LIN {X 0,Y 368.091,Z 174.068,A -85,B 0,C 180,E1 -12913.968,E2 -12913.968} C_VEL
LIN {X 0,Y 364.016,Z 163.404,A -85,B 0,C 180,E1 -12914.51,E2 -12914.51} C_VEL
LIN {X 0,Y 361.954,Z 153.4,A -85,B 0,C 180,E1 -12917.362,E2 -12917.362} C_VEL
LIN {X 0,Y 361.871,Z 153.409,A -85,B 0,C 180,E1 -12920.973,E2 -12920.973} C_VEL
LIN {X 0,Y 361.871,Z 153.409,A -85,B 0,C 180,E1 -12924.656,E2 -12924.656} C_VEL
LIN {X 0,Y 361.835,Z 153.411,A -85,B 0,C 180,E1 -12928.372,E2 -12928.372} C_VEL
LIN {X 0,Y 361.898,Z 153.403,A -85,B 0,C 180,E1 -12930.956,E2 -12930.956} C_VEL
LIN {X 0,Y 361.953,Z 153.4,A -85,B 0,C 180,E1 -12933.476,E2 -12933.476} C_VEL
LIN {X 0,Y 361.889,Z 153.41,A -85,B 0,C 180,E1 -12937.146,E2 -12937.146} C_VEL
LIN {X 0,Y 361.903,Z 153.406,A -85,B 0,C 180,E1 -12940.724,E2 -12940.724} C_VEL
LIN {X 0,Y 361.943,Z 153.398,A -85,B 0,C 180,E1 -12944.227,E2 -12944.227} C_VEL
LIN {X 0,Y 361.999,Z 153.388,A -85,B 0,C 180,E1 -12946.529,E2 -12946.529} C_VEL
LIN {X 0,Y 362.001,Z 153.389,A -85,B 0,C 180,E1 -12949.938,E2 -12949.938} C_VEL
LIN {X 0,Y 362.136,Z 153.373,A -85,B 0,C 180,E1 -12953.314,E2 -12953.314} C_VEL
LIN {X 0,Y 362.279,Z 153.352,A -85,B 0,C 180,E1 -12957.777,E2 -12957.777} C_VEL
LIN {X 0,Y 362.382,Z 153.337,A -85,B 0,C 180,E1 -12960.001,E2 -12960.001} C_VEL
LIN {X 0,Y 362.267,Z 153.352,A -85,B 0,C 180,E1 -12962.225,E2 -12962.225} C_VEL
LIN {X 0,Y 362.125,Z 153.37,A -85,B 0,C 180,E1 -12966.688,E2 -12966.688} C_VEL
LIN {X 0,Y 362.001,Z 153.384,A -85,B 0,C 180,E1 -12970.064,E2 -12970.064} C_VEL
LIN {X 0,Y 361.984,Z 153.397,A -85,B 0,C 180,E1 -12973.889,E2 -12973.889} C_VEL
LIN {X 0,Y 361.909,Z 153.405,A -85,B 0,C 180,E1 -12978.103,E2 -12978.103} C_VEL
LIN {X 0,Y 361.855,Z 153.403,A -85,B 0,C 180,E1 -12981.656,E2 -12981.656} C_VEL
LIN {X 0,Y 361.862,Z 153.407,A -85,B 0,C 180,E1 -12985.296,E2 -12985.296} C_VEL
LIN {X 0,Y 361.858,Z 153.411,A -85,B 0,C 180,E1 -12989.074,E2 -12989.074} C_VEL
LIN {X 0,Y 361.849,Z 153.412,A -85,B 0,C 180,E1 -12992.946,E2 -12992.946} C_VEL
LIN {X 0,Y 361.865,Z 153.41,A -85,B 0,C 180,E1 -12995.638,E2 -12995.638} C_VEL
LIN {X 0,Y 361.826,Z 153.414,A -85,B 0,C 180,E1 -12999.018,E2 -12999.018} C_VEL
LIN {X 0,Y 361.831,Z 153.419,A -85,B 0,C 180,E1 -13002.831,E2 -13002.831} C_VEL
LIN {X 0,Y 361.816,Z 153.419,A -85,B 0,C 180,E1 -13005.948,E2 -13005.948} C_VEL
LIN {X 0,Y 361.813,Z 153.419,A -85,B 0,C 180,E1 -13009.25,E2 -13009.25} C_VEL
LIN {X 0,Y 361.866,Z 153.403,A -85,B 0,C 180,E1 -13012.982,E2 -13012.982} C_VEL
LIN {X 0,Y 361.861,Z 153.408,A -85,B 0,C 180,E1 -13016.631,E2 -13016.631} C_VEL
LIN {X 0,Y 361.91,Z 153.464,A -85,B 0,C 180,E1 -13019.485,E2 -13019.485} C_VEL
LIN {X 0,Y 364.43,Z 165.067,A -85,B 0,C 180,E1 -13022.513,E2 -13022.513} C_VEL
LIN {X 0,Y 365.971,Z 173.011,A -85,B 0,C 180,E1 -13024.5,E2 -13024.5} C_VEL
LIN {X 0,Y 365.06,Z 184.322,A -85,B 0,C 180,E1 -13027.055,E2 -13027.055} C_VEL
LIN {X 0,Y 364.787,Z 186.723,A -85,B 0,C 180,E1 -13027.588,E2 -13027.588} C_VEL
LIN {X 0,Y 368.969,Z 210.144,A -85,B 0,C 180,E1 -13028.388,E2 -13028.388} C_VEL
LIN {X 0,Y 370.637,Z 222.589,A -85,B 0,C 180,E1 -13028.758,E2 -13028.758} C_VEL
LIN {X 0,Y 369.343,Z 296.316,A -85,B 0,C 180,E1 -13030.26,E2 -13030.26} C_VEL
LIN {X 0,Y 368.516,Z 309.974,A -85,B 0,C 180,E1 -13030.757,E2 -13030.757} C_VEL
LIN {X 0,Y 367.539,Z 322.813,A -85,B 0,C 180,E1 -13031.464,E2 -13031.464} C_VEL
LIN {X 0,Y 366.451,Z 335.344,A -85,B 0,C 180,E1 -13032.419,E2 -13032.419} C_VEL
LIN {X 0,Y 365.246,Z 346.544,A -85,B 0,C 180,E1 -13033.512,E2 -13033.512} C_VEL
LIN {X 0,Y 364.166,Z 356.855,A -85,B 0,C 180,E1 -13034.786,E2 -13034.786} C_VEL
LIN {X 0,Y 363.107,Z 366.602,A -85,B 0,C 180,E1 -13036.285,E2 -13036.285} C_VEL
LIN {X 0,Y 362.031,Z 375.393,A -85,B 0,C 180,E1 -13037.955,E2 -13037.955} C_VEL
LIN {X 0,Y 361.31,Z 382.419,A -85,B 0,C 180,E1 -13039.635,E2 -13039.635} C_VEL
LIN {X 0,Y 360.762,Z 388.878,A -85,B 0,C 180,E1 -13041.599,E2 -13041.599} C_VEL
LIN {X 0,Y 360.488,Z 393.134,A -85,B 0,C 180,E1 -13043.283,E2 -13043.283} C_VEL
LIN {X 0,Y 360.348,Z 395.396,A -85,B 0,C 180,E1 -13044.404,E2 -13044.404} C_VEL
LIN {X 0,Y 360.36,Z 397.178,A -85,B 0,C 180,E1 -13045.526,E2 -13045.526} C_VEL
LIN {X 0,Y 360.299,Z 399.5,A -85,B 0,C 180,E1 -13047.764,E2 -13047.764} C_VEL
LIN {X 0,Y 360.371,Z 400.07,A -85,B 0,C 180,E1 -13048.883,E2 -13048.883} C_VEL
LIN {X 0,Y 360.428,Z 400.201,A -85,B 0,C 180,E1 -13050,E2 -13050} C_VEL
LIN {X 0,Y 360.387,Z 399.931,A -85,B 0,C 180,E1 -13051.118,E2 -13051.118} C_VEL
LIN {X 0,Y 360.304,Z 398.214,A -85,B 0,C 180,E1 -13053.355,E2 -13053.355} C_VEL
LIN {X 0,Y 360.36,Z 396.702,A -85,B 0,C 180,E1 -13054.474,E2 -13054.474} C_VEL
LIN {X 0,Y 360.38,Z 394.055,A -85,B 0,C 180,E1 -13055.961,E2 -13055.961} C_VEL
LIN {X 0,Y 360.647,Z 389.498,A -85,B 0,C 180,E1 -13057.84,E2 -13057.84} C_VEL
LIN {X 0,Y 361.077,Z 383.159,A -85,B 0,C 180,E1 -13059.806,E2 -13059.806} C_VEL
LIN {X 0,Y 361.657,Z 376.253,A -85,B 0,C 180,E1 -13061.49,E2 -13061.49} C_VEL
LIN {X 0,Y 362.63,Z 367.626,A -85,B 0,C 180,E1 -13063.163,E2 -13063.163} C_VEL
LIN {X 0,Y 363.61,Z 357.664,A -85,B 0,C 180,E1 -13064.712,E2 -13064.712} C_VEL
LIN {X 0,Y 364.497,Z 347.838,A -85,B 0,C 180,E1 -13065.948,E2 -13065.948} C_VEL
LIN {X 0,Y 365.582,Z 336.839,A -85,B 0,C 180,E1 -13067.048,E2 -13067.048} C_VEL
LIN {X 0,Y 366.652,Z 324.514,A -85,B 0,C 180,E1 -13068.004,E2 -13068.004} C_VEL
LIN {X 0,Y 367.503,Z 312.873,A -85,B 0,C 180,E1 -13068.683,E2 -13068.683} C_VEL
LIN {X 0,Y 368.158,Z 300.549,A -85,B 0,C 180,E1 -13069.19,E2 -13069.19} C_VEL
LIN {X 0,Y 368.573,Z 285.008,A -85,B 0,C 180,E1 -13069.566,E2 -13069.566} C_VEL
LIN {X 0,Y 369.542,Z 221.072,A -85,B 0,C 180,E1 -13070.833,E2 -13070.833} C_VEL
LIN {X 0,Y 364.298,Z 187.546,A -85,B 0,C 180,E1 -13071.838,E2 -13071.838} C_VEL
LIN {X 0,Y 365.573,Z 174.668,A -85,B 0,C 180,E1 -13074.717,E2 -13074.717} C_VEL
LIN {X 0,Y 365.598,Z 171.805,A -85,B 0,C 180,E1 -13075.377,E2 -13075.377} C_VEL
LIN {X 0,Y 363.305,Z 160.054,A -85,B 0,C 180,E1 -13078.291,E2 -13078.291} C_VEL
LIN {X 0,Y 361.879,Z 153.41,A -85,B 0,C 180,E1 -13080.025,E2 -13080.025} C_VEL
LIN {X 0,Y 361.863,Z 153.41,A -85,B 0,C 180,E1 -13083.369,E2 -13083.369} C_VEL
LIN {X 0,Y 361.869,Z 153.407,A -85,B 0,C 180,E1 -13087.018,E2 -13087.018} C_VEL
LIN {X 0,Y 361.816,Z 153.413,A -85,B 0,C 180,E1 -13090.751,E2 -13090.751} C_VEL
LIN {X 0,Y 361.816,Z 153.412,A -85,B 0,C 180,E1 -13094.369,E2 -13094.369} C_VEL
LIN {X 0,Y 361.834,Z 153.413,A -85,B 0,C 180,E1 -13097.569,E2 -13097.569} C_VEL
LIN {X 0,Y 361.849,Z 153.41,A -85,B 0,C 180,E1 -13101.572,E2 -13101.572} C_VEL
LIN {X 0,Y 361.875,Z 153.407,A -85,B 0,C 180,E1 -13104.656,E2 -13104.656} C_VEL
LIN {X 0,Y 361.842,Z 153.41,A -85,B 0,C 180,E1 -13108.37,E2 -13108.37} C_VEL
LIN {X 0,Y 361.871,Z 153.411,A -85,B 0,C 180,E1 -13110.952,E2 -13110.952} C_VEL
LIN {X 0,Y 361.886,Z 153.408,A -85,B 0,C 180,E1 -13114.706,E2 -13114.706} C_VEL
LIN {X 0,Y 361.859,Z 153.409,A -85,B 0,C 180,E1 -13118.344,E2 -13118.344} C_VEL
LIN {X 0,Y 361.909,Z 153.402,A -85,B 0,C 180,E1 -13122.092,E2 -13122.092} C_VEL
LIN {X 0,Y 361.985,Z 153.393,A -85,B 0,C 180,E1 -13126.112,E2 -13126.112} C_VEL
LIN {X 0,Y 362.003,Z 153.39,A -85,B 0,C 180,E1 -13129.936,E2 -13129.936} C_VEL
LIN {X 0,Y 362.126,Z 153.374,A -85,B 0,C 180,E1 -13133.312,E2 -13133.312} C_VEL
LIN {X 0,Y 362.268,Z 153.357,A -85,B 0,C 180,E1 -13137.775,E2 -13137.775} C_VEL
LIN {X 0,Y 362.179,Z 153.367,A -85,B 0,C 180,E1 -13141.111,E2 -13141.111} C_VEL
LIN {X 0,Y 362.267,Z 153.362,A -85,B 0,C 180,E1 -13142.223,E2 -13142.223} C_VEL
LIN {X 0,Y 362.122,Z 153.375,A -85,B 0,C 180,E1 -13146.686,E2 -13146.686} C_VEL
LIN {X 0,Y 361.997,Z 153.395,A -85,B 0,C 180,E1 -13150.062,E2 -13150.062} C_VEL
LIN {X 0,Y 361.982,Z 153.398,A -85,B 0,C 180,E1 -13153.886,E2 -13153.886} C_VEL
LIN {X 0,Y 361.885,Z 153.407,A -85,B 0,C 180,E1 -13158.102,E2 -13158.102} C_VEL
LIN {X 0,Y 361.853,Z 153.413,A -85,B 0,C 180,E1 -13161.654,E2 -13161.654} C_VEL
LIN {X 0,Y 361.852,Z 153.411,A -85,B 0,C 180,E1 -13165.295,E2 -13165.295} C_VEL
LIN {X 0,Y 361.855,Z 153.409,A -85,B 0,C 180,E1 -13169.072,E2 -13169.072} C_VEL
LIN {X 0,Y 361.846,Z 153.41,A -85,B 0,C 180,E1 -13172.944,E2 -13172.944} C_VEL
LIN {X 0,Y 361.865,Z 153.41,A -85,B 0,C 180,E1 -13175.636,E2 -13175.636} C_VEL
LIN {X 0,Y 361.823,Z 153.415,A -85,B 0,C 180,E1 -13179.017,E2 -13179.017} C_VEL
LIN {X 0,Y 361.827,Z 153.413,A -85,B 0,C 180,E1 -13182.829,E2 -13182.829} C_VEL
LIN {X 0,Y 361.809,Z 153.413,A -85,B 0,C 180,E1 -13185.946,E2 -13185.946} C_VEL
LIN {X 0,Y 361.808,Z 153.417,A -85,B 0,C 180,E1 -13189.248,E2 -13189.248} C_VEL
LIN {X 0,Y 361.858,Z 153.413,A -85,B 0,C 180,E1 -13192.98,E2 -13192.98} C_VEL
LIN {X 0,Y 361.852,Z 153.411,A -85,B 0,C 180,E1 -13196.63,E2 -13196.63} C_VEL
LIN {X 0,Y 361.85,Z 153.408,A -85,B 0,C 180,E1 -13199.669,E2 -13199.669} C_VEL
LIN {X 0,Y 361.849,Z 153.408,A -85,B 0,C 180,E1 -13203.466,E2 -13203.466} C_VEL
LIN {X 0,Y 361.855,Z 153.409,A -85,B 0,C 180,E1 -13207.142,E2 -13207.142} C_VEL
LIN {X 0,Y 361.847,Z 153.413,A -85,B 0,C 180,E1 -13210.72,E2 -13210.72} C_VEL
LIN {X 0,Y 361.888,Z 153.407,A -85,B 0,C 180,E1 -13214.223,E2 -13214.223} C_VEL
LIN {X 0,Y 361.992,Z 153.395,A -85,B 0,C 180,E1 -13216.527,E2 -13216.527} C_VEL
LIN {X 0,Y 361.987,Z 153.393,A -85,B 0,C 180,E1 -13219.936,E2 -13219.936} C_VEL
LIN {X 0,Y 362.114,Z 153.375,A -85,B 0,C 180,E1 -13223.312,E2 -13223.312} C_VEL
LIN {X 0,Y 362.189,Z 153.39,A -85,B 0,C 180,E1 -13227.567,E2 -13227.567} C_VEL
LIN {X 0,Y 363.918,Z 163.048,A -85,B 0,C 180,E1 -13230.214,E2 -13230.214} C_VEL
LIN {X 0,Y 366.792,Z 172.146,A -85,B 0,C 180,E1 -13230.576,E2 -13230.576} C_VEL
LIN {X 0,Y 370.036,Z 187.803,A -85,B 0,C 180,E1 -13231.088,E2 -13231.088} C_VEL
LIN {X 0,Y 368.599,Z 270.026,A -85,B 0,C 180,E1 -13232.732,E2 -13232.732} C_VEL
LIN {X 0,Y 368.077,Z 282.649,A -85,B 0,C 180,E1 -13233.181,E2 -13233.181} C_VEL
LIN {X 0,Y 367.405,Z 296.158,A -85,B 0,C 180,E1 -13233.907,E2 -13233.907} C_VEL
LIN {X 0,Y 366.547,Z 308.584,A -85,B 0,C 180,E1 -13234.834,E2 -13234.834} C_VEL
LIN {X 0,Y 365.609,Z 319.937,A -85,B 0,C 180,E1 -13235.93,E2 -13235.93} C_VEL
LIN {X 0,Y 364.589,Z 330.413,A -85,B 0,C 180,E1 -13237.198,E2 -13237.198} C_VEL
LIN {X 0,Y 363.606,Z 339.787,A -85,B 0,C 180,E1 -13238.615,E2 -13238.615} C_VEL
LIN {X 0,Y 362.596,Z 348.911,A -85,B 0,C 180,E1 -13240.328,E2 -13240.328} C_VEL
LIN {X 0,Y 361.859,Z 356.191,A -85,B 0,C 180,E1 -13242.051,E2 -13242.051} C_VEL
LIN {X 0,Y 361.331,Z 361.133,A -85,B 0,C 180,E1 -13243.497,E2 -13243.497} C_VEL
LIN {X 0,Y 360.906,Z 365.868,A -85,B 0,C 180,E1 -13245.241,E2 -13245.241} C_VEL
LIN {X 0,Y 360.511,Z 369.794,A -85,B 0,C 180,E1 -13247.213,E2 -13247.213} C_VEL
LIN {X 0,Y 360.275,Z 372.567,A -85,B 0,C 180,E1 -13249.367,E2 -13249.367} C_VEL
LIN {X 0,Y 360.162,Z 373.608,A -85,B 0,C 180,E1 -13251.025,E2 -13251.025} C_VEL
LIN {X 0,Y 360.2,Z 373.839,A -85,B 0,C 180,E1 -13252.969,E2 -13252.969} C_VEL
LIN {X 0,Y 360.25,Z 373.344,A -85,B 0,C 180,E1 -13254.185,E2 -13254.185} C_VEL
LIN {X 0,Y 360.427,Z 371.817,A -85,B 0,C 180,E1 -13255.879,E2 -13255.879} C_VEL
LIN {X 0,Y 359.904,Z 370.713,A -85,B 0,C 180,E1 -13256.798,E2 -13256.798} C_VEL
LIN {X 0,Y 357.295,Z 368.435,A -85,B 0,C 180,E1 -13258.286,E2 -13258.286} C_VEL
LIN {X 0,Y 355.141,Z 366.13,A -85,B 0,C 180,E1 -13259.465,E2 -13259.465} C_VEL
LIN {X 0,Y 354.359,Z 364.018,A -85,B 0,C 180,E1 -13260.351,E2 -13260.351} C_VEL
LIN {X 0,Y 354.374,Z 363.21,A -85,B 0,C 180,E1 -13260.644,E2 -13260.644} C_VEL
LIN {X 0,Y 355.171,Z 356.911,A -85,B 0,C 180,E1 -13262.63,E2 -13262.63} C_VEL
LIN {X 0,Y 356.081,Z 349.885,A -85,B 0,C 180,E1 -13264.36,E2 -13264.36} C_VEL
LIN {X 0,Y 357.002,Z 342.397,A -85,B 0,C 180,E1 -13265.85,E2 -13265.85} C_VEL
LIN {X 0,Y 358.233,Z 332.376,A -85,B 0,C 180,E1 -13267.458,E2 -13267.458} C_VEL
LIN {X 0,Y 359.421,Z 322.449,A -85,B 0,C 180,E1 -13268.735,E2 -13268.735} C_VEL
LIN {X 0,Y 360.491,Z 311.509,A -85,B 0,C 180,E1 -13269.86,E2 -13269.86} C_VEL
LIN {X 0,Y 361.527,Z 299.931,A -85,B 0,C 180,E1 -13270.789,E2 -13270.789} C_VEL
LIN {X 0,Y 362.271,Z 287.523,A -85,B 0,C 180,E1 -13271.547,E2 -13271.547} C_VEL
LIN {X 0,Y 362.862,Z 274.421,A -85,B 0,C 180,E1 -13272.092,E2 -13272.092} C_VEL
LIN {X 0,Y 363.358,Z 256.473,A -85,B 0,C 180,E1 -13272.513,E2 -13272.513} C_VEL
LIN {X 0,Y 364.736,Z 190.027,A -85,B 0,C 180,E1 -13273.854,E2 -13273.854} C_VEL
LIN {X 0,Y 361.911,Z 176.606,A -85,B 0,C 180,E1 -13274.345,E2 -13274.345} C_VEL
LIN {X 0,Y 356.896,Z 163.731,A -85,B 0,C 180,E1 -13275.013,E2 -13275.013} C_VEL
LIN {X 0,Y 354.874,Z 154.284,A -85,B 0,C 180,E1 -13277.754,E2 -13277.754} C_VEL
LIN {X 0,Y 354.833,Z 154.286,A -85,B 0,C 180,E1 -13280.67,E2 -13280.67} C_VEL
LIN {X 0,Y 354.819,Z 154.289,A -85,B 0,C 180,E1 -13284.302,E2 -13284.302} C_VEL
LIN {X 0,Y 354.784,Z 154.292,A -85,B 0,C 180,E1 -13287.668,E2 -13287.668} C_VEL
LIN {X 0,Y 354.866,Z 154.277,A -85,B 0,C 180,E1 -13290.622,E2 -13290.622} C_VEL
LIN {X 0,Y 354.898,Z 154.279,A -85,B 0,C 180,E1 -13294.174,E2 -13294.174} C_VEL
LIN {X 0,Y 354.834,Z 154.286,A -85,B 0,C 180,E1 -13297.895,E2 -13297.895} C_VEL
LIN {X 0,Y 354.889,Z 154.275,A -85,B 0,C 180,E1 -13301.909,E2 -13301.909} C_VEL
LIN {X 0,Y 354.943,Z 154.267,A -85,B 0,C 180,E1 -13305.982,E2 -13305.982} C_VEL
LIN {X 0,Y 354.957,Z 154.267,A -85,B 0,C 180,E1 -13309.736,E2 -13309.736} C_VEL
LIN {X 0,Y 355.1,Z 154.25,A -85,B 0,C 180,E1 -13313.181,E2 -13313.181} C_VEL
LIN {X 0,Y 355.242,Z 154.229,A -85,B 0,C 180,E1 -13317.733,E2 -13317.733} C_VEL
LIN {X 0,Y 355.333,Z 154.215,A -85,B 0,C 180,E1 -13320.001,E2 -13320.001} C_VEL
LIN {X 0,Y 355.229,Z 154.229,A -85,B 0,C 180,E1 -13322.269,E2 -13322.269} C_VEL
LIN {X 0,Y 355.091,Z 154.247,A -85,B 0,C 180,E1 -13326.821,E2 -13326.821} C_VEL
LIN {X 0,Y 354.957,Z 154.259,A -85,B 0,C 180,E1 -13330.266,E2 -13330.266} C_VEL
LIN {X 0,Y 354.929,Z 154.275,A -85,B 0,C 180,E1 -13334.009,E2 -13334.009} C_VEL
LIN {X 0,Y 354.865,Z 154.282,A -85,B 0,C 180,E1 -13338.079,E2 -13338.079} C_VEL
LIN {X 0,Y 354.808,Z 154.283,A -85,B 0,C 180,E1 -13342.109,E2 -13342.109} C_VEL
LIN {X 0,Y 354.801,Z 154.281,A -85,B 0,C 180,E1 -13345.836,E2 -13345.836} C_VEL
LIN {X 0,Y 354.795,Z 154.285,A -85,B 0,C 180,E1 -13349.685,E2 -13349.685} C_VEL
LIN {X 0,Y 354.788,Z 154.29,A -85,B 0,C 180,E1 -13352.334,E2 -13352.334} C_VEL
LIN {X 0,Y 354.82,Z 154.288,A -85,B 0,C 180,E1 -13355.699,E2 -13355.699} C_VEL
LIN {X 0,Y 354.771,Z 154.297,A -85,B 0,C 180,E1 -13359.413,E2 -13359.413} C_VEL
LIN {X 0,Y 354.783,Z 154.298,A -85,B 0,C 180,E1 -13362.866,E2 -13362.866} C_VEL
LIN {X 0,Y 354.765,Z 154.298,A -85,B 0,C 180,E1 -13366.103,E2 -13366.103} C_VEL
LIN {X 0,Y 354.765,Z 154.297,A -85,B 0,C 180,E1 -13369.176,E2 -13369.176} C_VEL
LIN {X 0,Y 354.803,Z 154.288,A -85,B 0,C 180,E1 -13372.405,E2 -13372.405} C_VEL
LIN {X 0,Y 354.814,Z 154.289,A -85,B 0,C 180,E1 -13374.941,E2 -13374.941} C_VEL
LIN {X 0,Y 354.793,Z 154.288,A -85,B 0,C 180,E1 -13378.407,E2 -13378.407} C_VEL
LIN {X 0,Y 354.842,Z 154.331,A -85,B 0,C 180,E1 -13379.051,E2 -13379.051} C_VEL
LIN {X 0,Y 357.162,Z 164.602,A -85,B 0,C 180,E1 -13381.819,E2 -13381.819} C_VEL
LIN {X 0,Y 359.121,Z 175.083,A -85,B 0,C 180,E1 -13384.498,E2 -13384.498} C_VEL
LIN {X 0,Y 358.055,Z 186.716,A -85,B 0,C 180,E1 -13387.128,E2 -13387.128} C_VEL
LIN {X 0,Y 362.525,Z 211.613,A -85,B 0,C 180,E1 -13387.991,E2 -13387.991} C_VEL
LIN {X 0,Y 364.09,Z 223.708,A -85,B 0,C 180,E1 -13388.357,E2 -13388.357} C_VEL
LIN {X 0,Y 362.74,Z 295.788,A -85,B 0,C 180,E1 -13389.848,E2 -13389.848} C_VEL
LIN {X 0,Y 361.925,Z 309.526,A -85,B 0,C 180,E1 -13390.356,E2 -13390.356} C_VEL
LIN {X 0,Y 360.916,Z 321.914,A -85,B 0,C 180,E1 -13391.038,E2 -13391.038} C_VEL
LIN {X 0,Y 359.832,Z 333.796,A -85,B 0,C 180,E1 -13391.937,E2 -13391.937} C_VEL
LIN {X 0,Y 358.558,Z 345.229,A -85,B 0,C 180,E1 -13393.049,E2 -13393.049} C_VEL
LIN {X 0,Y 357.418,Z 355.6,A -85,B 0,C 180,E1 -13394.319,E2 -13394.319} C_VEL
LIN {X 0,Y 356.353,Z 364.852,A -85,B 0,C 180,E1 -13395.728,E2 -13395.728} C_VEL
LIN {X 0,Y 355.259,Z 373.891,A -85,B 0,C 180,E1 -13397.431,E2 -13397.431} C_VEL
LIN {X 0,Y 354.388,Z 381.186,A -85,B 0,C 180,E1 -13399.141,E2 -13399.141} C_VEL
LIN {X 0,Y 353.855,Z 387.036,A -85,B 0,C 180,E1 -13400.858,E2 -13400.858} C_VEL
LIN {X 0,Y 353.466,Z 391.652,A -85,B 0,C 180,E1 -13402.575,E2 -13402.575} C_VEL
LIN {X 0,Y 353.284,Z 395.175,A -85,B 0,C 180,E1 -13404.292,E2 -13404.292} C_VEL
LIN {X 0,Y 353.27,Z 396.946,A -85,B 0,C 180,E1 -13405.436,E2 -13405.436} C_VEL
LIN {X 0,Y 353.224,Z 398.299,A -85,B 0,C 180,E1 -13406.578,E2 -13406.578} C_VEL
LIN {X 0,Y 353.271,Z 399.816,A -85,B 0,C 180,E1 -13408.86,E2 -13408.86} C_VEL
LIN {X 0,Y 353.332,Z 399.938,A -85,B 0,C 180,E1 -13410,E2 -13410} C_VEL
LIN {X 0,Y 353.287,Z 399.661,A -85,B 0,C 180,E1 -13411.14,E2 -13411.14} C_VEL
LIN {X 0,Y 353.225,Z 397.929,A -85,B 0,C 180,E1 -13413.422,E2 -13413.422} C_VEL
LIN {X 0,Y 353.27,Z 396.405,A -85,B 0,C 180,E1 -13414.564,E2 -13414.564} C_VEL
LIN {X 0,Y 353.335,Z 393.322,A -85,B 0,C 180,E1 -13416.28,E2 -13416.28} C_VEL
LIN {X 0,Y 353.573,Z 389.168,A -85,B 0,C 180,E1 -13417.998,E2 -13417.998} C_VEL
LIN {X 0,Y 354.055,Z 382.812,A -85,B 0,C 180,E1 -13420.003,E2 -13420.003} C_VEL
LIN {X 0,Y 354.663,Z 375.885,A -85,B 0,C 180,E1 -13421.719,E2 -13421.719} C_VEL
LIN {X 0,Y 355.656,Z 367.22,A -85,B 0,C 180,E1 -13423.426,E2 -13423.426} C_VEL
LIN {X 0,Y 356.605,Z 358.323,A -85,B 0,C 180,E1 -13424.845,E2 -13424.845} C_VEL
LIN {X 0,Y 357.509,Z 348.548,A -85,B 0,C 180,E1 -13426.122,E2 -13426.122} C_VEL
LIN {X 0,Y 358.628,Z 337.858,A -85,B 0,C 180,E1 -13427.242,E2 -13427.242} C_VEL
LIN {X 0,Y 359.718,Z 325.882,A -85,B 0,C 180,E1 -13428.216,E2 -13428.216} C_VEL
LIN {X 0,Y 360.691,Z 313.433,A -85,B 0,C 180,E1 -13428.975,E2 -13428.975} C_VEL
LIN {X 0,Y 361.397,Z 300.561,A -85,B 0,C 180,E1 -13429.527,E2 -13429.527} C_VEL
LIN {X 0,Y 361.836,Z 286.962,A -85,B 0,C 180,E1 -13429.871,E2 -13429.871} C_VEL
LIN {X 0,Y 362.851,Z 222.052,A -85,B 0,C 180,E1 -13431.181,E2 -13431.181} C_VEL
LIN {X 0,Y 357.747,Z 189.335,A -85,B 0,C 180,E1 -13432.175,E2 -13432.175} C_VEL
LIN {X 0,Y 357.447,Z 187.262,A -85,B 0,C 180,E1 -13432.255,E2 -13432.255} C_VEL
LIN {X 0,Y 358.643,Z 175.582,A -85,B 0,C 180,E1 -13434.918,E2 -13434.918} C_VEL
LIN {X 0,Y 358.38,Z 171.625,A -85,B 0,C 180,E1 -13435.87,E2 -13435.87} C_VEL
LIN {X 0,Y 356.008,Z 159.615,A -85,B 0,C 180,E1 -13438.925,E2 -13438.925} C_VEL
LIN {X 0,Y 354.843,Z 154.288,A -85,B 0,C 180,E1 -13440.335,E2 -13440.335} C_VEL
LIN {X 0,Y 354.811,Z 154.29,A -85,B 0,C 180,E1 -13443.702,E2 -13443.702} C_VEL
LIN {X 0,Y 354.8,Z 154.286,A -85,B 0,C 180,E1 -13446.46,E2 -13446.46} C_VEL
LIN {X 0,Y 354.773,Z 154.296,A -85,B 0,C 180,E1 -13449.412,E2 -13449.412} C_VEL
LIN {X 0,Y 354.787,Z 154.289,A -85,B 0,C 180,E1 -13452.866,E2 -13452.866} C_VEL
LIN {X 0,Y 354.767,Z 154.29,A -85,B 0,C 180,E1 -13456.103,E2 -13456.103} C_VEL
LIN {X 0,Y 354.771,Z 154.296,A -85,B 0,C 180,E1 -13459.176,E2 -13459.176} C_VEL
LIN {X 0,Y 354.805,Z 154.286,A -85,B 0,C 180,E1 -13462.404,E2 -13462.404} C_VEL
LIN {X 0,Y 354.814,Z 154.289,A -85,B 0,C 180,E1 -13464.94,E2 -13464.94} C_VEL
LIN {X 0,Y 354.798,Z 154.288,A -85,B 0,C 180,E1 -13468.405,E2 -13468.405} C_VEL
LIN {X 0,Y 354.805,Z 154.286,A -85,B 0,C 180,E1 -13471.614,E2 -13471.614} C_VEL
LIN {X 0,Y 354.839,Z 154.281,A -85,B 0,C 180,E1 -13475.657,E2 -13475.657} C_VEL
LIN {X 0,Y 354.829,Z 154.285,A -85,B 0,C 180,E1 -13479.112,E2 -13479.112} C_VEL
LIN {X 0,Y 354.856,Z 154.285,A -85,B 0,C 180,E1 -13482.717,E2 -13482.717} C_VEL
LIN {X 0,Y 354.945,Z 154.271,A -85,B 0,C 180,E1 -13486.254,E2 -13486.254} C_VEL
LIN {X 0,Y 354.96,Z 154.267,A -85,B 0,C 180,E1 -13489.734,E2 -13489.734} C_VEL
LIN {X 0,Y 355.092,Z 154.25,A -85,B 0,C 180,E1 -13493.179,E2 -13493.179} C_VEL
LIN {X 0,Y 355.231,Z 154.234,A -85,B 0,C 180,E1 -13497.731,E2 -13497.731} C_VEL
LIN {X 0,Y 355.15,Z 154.243,A -85,B 0,C 180,E1 -13501.133,E2 -13501.133} C_VEL
LIN {X 0,Y 355.229,Z 154.238,A -85,B 0,C 180,E1 -13502.267,E2 -13502.267} C_VEL
LIN {X 0,Y 355.088,Z 154.251,A -85,B 0,C 180,E1 -13506.819,E2 -13506.819} C_VEL
LIN {X 0,Y 354.954,Z 154.27,A -85,B 0,C 180,E1 -13510.264,E2 -13510.264} C_VEL
LIN {X 0,Y 354.925,Z 154.276,A -85,B 0,C 180,E1 -13514.004,E2 -13514.004} C_VEL
LIN {X 0,Y 354.843,Z 154.284,A -85,B 0,C 180,E1 -13518.067,E2 -13518.067} C_VEL
LIN {X 0,Y 354.806,Z 154.288,A -85,B 0,C 180,E1 -13522.107,E2 -13522.107} C_VEL
LIN {X 0,Y 354.795,Z 154.291,A -85,B 0,C 180,E1 -13525.834,E2 -13525.834} C_VEL
LIN {X 0,Y 354.795,Z 154.291,A -85,B 0,C 180,E1 -13529.683,E2 -13529.683} C_VEL
LIN {X 0,Y 354.785,Z 154.288,A -85,B 0,C 180,E1 -13532.332,E2 -13532.332} C_VEL
LIN {X 0,Y 354.819,Z 154.287,A -85,B 0,C 180,E1 -13535.698,E2 -13535.698} C_VEL
LIN {X 0,Y 354.765,Z 154.295,A -85,B 0,C 180,E1 -13539.411,E2 -13539.411} C_VEL
LIN {X 0,Y 354.78,Z 154.292,A -85,B 0,C 180,E1 -13542.865,E2 -13542.865} C_VEL
LIN {X 0,Y 354.759,Z 154.291,A -85,B 0,C 180,E1 -13546.102,E2 -13546.102} C_VEL
LIN {X 0,Y 354.762,Z 154.296,A -85,B 0,C 180,E1 -13549.175,E2 -13549.175} C_VEL
LIN {X 0,Y 354.795,Z 154.288,A -85,B 0,C 180,E1 -13552.403,E2 -13552.403} C_VEL
LIN {X 0,Y 354.804,Z 154.292,A -85,B 0,C 180,E1 -13554.939,E2 -13554.939} C_VEL
LIN {X 0,Y 354.788,Z 154.29,A -85,B 0,C 180,E1 -13558.404,E2 -13558.404} C_VEL
LIN {X 0,Y 354.791,Z 154.287,A -85,B 0,C 180,E1 -13561.613,E2 -13561.613} C_VEL
LIN {X 0,Y 354.797,Z 154.287,A -85,B 0,C 180,E1 -13565.419,E2 -13565.419} C_VEL
LIN {X 0,Y 354.814,Z 154.286,A -85,B 0,C 180,E1 -13569.112,E2 -13569.112} C_VEL
LIN {X 0,Y 354.844,Z 154.284,A -85,B 0,C 180,E1 -13572.717,E2 -13572.717} C_VEL
LIN {X 0,Y 354.932,Z 154.274,A -85,B 0,C 180,E1 -13576.254,E2 -13576.254} C_VEL
LIN {X 0,Y 354.944,Z 154.269,A -85,B 0,C 180,E1 -13579.735,E2 -13579.735} C_VEL
LIN {X 0,Y 355.079,Z 154.251,A -85,B 0,C 180,E1 -13583.179,E2 -13583.179} C_VEL
LIN {X 0,Y 355.143,Z 154.445,A -85,B 0,C 180,E1 -13587.306,E2 -13587.306} C_VEL
LIN {X 0,Y 356.834,Z 163.204,A -85,B 0,C 180,E1 -13589.778,E2 -13589.778} C_VEL
LIN {X 0,Y 360.478,Z 174.747,A -85,B 0,C 180,E1 -13590.26,E2 -13590.26} C_VEL
LIN {X 0,Y 363.371,Z 188.971,A -85,B 0,C 180,E1 -13590.734,E2 -13590.734} C_VEL
LIN {X 0,Y 361.853,Z 270.681,A -85,B 0,C 180,E1 -13592.4,E2 -13592.4} C_VEL
LIN {X 0,Y 361.306,Z 283.182,A -85,B 0,C 180,E1 -13592.857,E2 -13592.857} C_VEL
LIN {X 0,Y 360.647,Z 296.048,A -85,B 0,C 180,E1 -13593.561,E2 -13593.561} C_VEL
LIN {X 0,Y 359.777,Z 308.332,A -85,B 0,C 180,E1 -13594.481,E2 -13594.481} C_VEL
LIN {X 0,Y 358.752,Z 320.005,A -85,B 0,C 180,E1 -13595.621,E2 -13595.621} C_VEL
LIN {X 0,Y 357.717,Z 330.512,A -85,B 0,C 180,E1 -13596.911,E2 -13596.911} C_VEL
LIN {X 0,Y 356.79,Z 339.087,A -85,B 0,C 180,E1 -13598.21,E2 -13598.21} C_VEL
LIN {X 0,Y 355.714,Z 348.328,A -85,B 0,C 180,E1 -13599.945,E2 -13599.945} C_VEL
LIN {X 0,Y 354.923,Z 355.829,A -85,B 0,C 180,E1 -13601.71,E2 -13601.71} C_VEL
LIN {X 0,Y 354.229,Z 361.979,A -85,B 0,C 180,E1 -13603.553,E2 -13603.553} C_VEL
LIN {X 0,Y 353.751,Z 367.061,A -85,B 0,C 180,E1 -13605.557,E2 -13605.557} C_VEL
LIN {X 0,Y 353.387,Z 370.393,A -85,B 0,C 180,E1 -13607.356,E2 -13607.356} C_VEL
LIN {X 0,Y 353.239,Z 372.041,A -85,B 0,C 180,E1 -13608.562,E2 -13608.562} C_VEL
LIN {X 0,Y 353.089,Z 373.77,A -85,B 0,C 180,E1 -13610.694,E2 -13610.694} C_VEL
LIN {X 0,Y 353.062,Z 374.186,A -85,B 0,C 180,E1 -13612.223,E2 -13612.223} C_VEL
LIN {X 0,Y 353.147,Z 373.855,A -85,B 0,C 180,E1 -13613.734,E2 -13613.734} C_VEL
LIN {X 0,Y 353.374,Z 372.17,A -85,B 0,C 180,E1 -13615.947,E2 -13615.947} C_VEL
LIN {X 0,Y 353.681,Z 369.479,A -85,B 0,C 180,E1 -13617.838,E2 -13617.838} C_VEL
LIN {X 0,Y 354.085,Z 365.524,A -85,B 0,C 180,E1 -13619.749,E2 -13619.749} C_VEL
LIN {X 0,Y 354.374,Z 363.21,A -85,B 0,C 180,E1 -13620.644,E2 -13620.644} C_VEL
LIN {X 0,Y 354.033,Z 360.767,A -85,B 0,C 180,E1 -13621.511,E2 -13621.511} C_VEL
LIN {X 0,Y 351.783,Z 356.457,A -85,B 0,C 180,E1 -13622.915,E2 -13622.915} C_VEL
LIN {X 0,Y 349.629,Z 351.554,A -85,B 0,C 180,E1 -13624.28,E2 -13624.28} C_VEL
LIN {X 0,Y 349.438,Z 348.123,A -85,B 0,C 180,E1 -13625.072,E2 -13625.072} C_VEL
LIN {X 0,Y 350.599,Z 339.597,A -85,B 0,C 180,E1 -13626.697,E2 -13626.697} C_VEL
LIN {X 0,Y 351.703,Z 330.519,A -85,B 0,C 180,E1 -13628.095,E2 -13628.095} C_VEL
LIN {X 0,Y 352.985,Z 320.146,A -85,B 0,C 180,E1 -13629.379,E2 -13629.379} C_VEL
LIN {X 0,Y 353.943,Z 310.231,A -85,B 0,C 180,E1 -13630.377,E2 -13630.377} C_VEL
LIN {X 0,Y 355.003,Z 298.45,A -85,B 0,C 180,E1 -13631.309,E2 -13631.309} C_VEL
LIN {X 0,Y 355.781,Z 285.66,A -85,B 0,C 180,E1 -13632.06,E2 -13632.06} C_VEL
LIN {X 0,Y 356.346,Z 272.471,A -85,B 0,C 180,E1 -13632.581,E2 -13632.581} C_VEL
LIN {X 0,Y 357.258,Z 233.094,A -85,B 0,C 180,E1 -13633.428,E2 -13633.428} C_VEL
LIN {X 0,Y 358.118,Z 190.113,A -85,B 0,C 180,E1 -13634.318,E2 -13634.318} C_VEL
LIN {X 0,Y 355.582,Z 178.575,A -85,B 0,C 180,E1 -13634.761,E2 -13634.761} C_VEL
LIN {X 0,Y 349.773,Z 164.037,A -85,B 0,C 180,E1 -13635.545,E2 -13635.545} C_VEL
LIN {X 0,Y 347.818,Z 155.16,A -85,B 0,C 180,E1 -13638.219,E2 -13638.219} C_VEL
LIN {X 0,Y 347.773,Z 155.174,A -85,B 0,C 180,E1 -13642.012,E2 -13642.012} C_VEL
LIN {X 0,Y 347.741,Z 155.173,A -85,B 0,C 180,E1 -13645.537,E2 -13645.537} C_VEL
LIN {X 0,Y 347.761,Z 155.166,A -85,B 0,C 180,E1 -13649.655,E2 -13649.655} C_VEL
LIN {X 0,Y 347.85,Z 155.155,A -85,B 0,C 180,E1 -13652.746,E2 -13652.746} C_VEL
LIN {X 0,Y 347.787,Z 155.161,A -85,B 0,C 180,E1 -13656.163,E2 -13656.163} C_VEL
LIN {X 0,Y 347.811,Z 155.16,A -85,B 0,C 180,E1 -13659.91,E2 -13659.91} C_VEL
LIN {X 0,Y 347.832,Z 155.157,A -85,B 0,C 180,E1 -13663.569,E2 -13663.569} C_VEL
LIN {X 0,Y 347.89,Z 155.145,A -85,B 0,C 180,E1 -13667.162,E2 -13667.162} C_VEL
LIN {X 0,Y 347.935,Z 155.137,A -85,B 0,C 180,E1 -13670.702,E2 -13670.702} C_VEL
LIN {X 0,Y 348.051,Z 155.129,A -85,B 0,C 180,E1 -13674.206,E2 -13674.206} C_VEL
LIN {X 0,Y 348.204,Z 155.105,A -85,B 0,C 180,E1 -13677.687,E2 -13677.687} C_VEL
LIN {X 0,Y 348.284,Z 155.092,A -85,B 0,C 180,E1 -13680.001,E2 -13680.001} C_VEL
LIN {X 0,Y 348.191,Z 155.106,A -85,B 0,C 180,E1 -13682.315,E2 -13682.315} C_VEL
LIN {X 0,Y 348.057,Z 155.122,A -85,B 0,C 180,E1 -13686.96,E2 -13686.96} C_VEL
LIN {X 0,Y 347.898,Z 155.136,A -85,B 0,C 180,E1 -13690.476,E2 -13690.476} C_VEL
LIN {X 0,Y 347.901,Z 155.149,A -85,B 0,C 180,E1 -13694.151,E2 -13694.151} C_VEL
LIN {X 0,Y 347.811,Z 155.16,A -85,B 0,C 180,E1 -13698.25,E2 -13698.25} C_VEL
LIN {X 0,Y 347.765,Z 155.157,A -85,B 0,C 180,E1 -13701.625,E2 -13701.625} C_VEL
LIN {X 0,Y 347.739,Z 155.168,A -85,B 0,C 180,E1 -13705.115,E2 -13705.115} C_VEL
LIN {X 0,Y 347.731,Z 155.17,A -85,B 0,C 180,E1 -13707.702,E2 -13707.702} C_VEL
LIN {X 0,Y 347.738,Z 155.16,A -85,B 0,C 180,E1 -13710.35,E2 -13710.35} C_VEL
LIN {X 0,Y 347.75,Z 155.161,A -85,B 0,C 180,E1 -13714.044,E2 -13714.044} C_VEL
LIN {X 0,Y 347.756,Z 155.164,A -85,B 0,C 180,E1 -13717.322,E2 -13717.322} C_VEL
LIN {X 0,Y 347.698,Z 155.175,A -85,B 0,C 180,E1 -13720.303,E2 -13720.303} C_VEL
LIN {X 0,Y 347.723,Z 155.172,A -85,B 0,C 180,E1 -13723.409,E2 -13723.409} C_VEL
LIN {X 0,Y 347.725,Z 155.174,A -85,B 0,C 180,E1 -13726.687,E2 -13726.687} C_VEL
LIN {X 0,Y 347.703,Z 155.177,A -85,B 0,C 180,E1 -13730.183,E2 -13730.183} C_VEL
LIN {X 0,Y 347.759,Z 155.163,A -85,B 0,C 180,E1 -13732.679,E2 -13732.679} C_VEL
LIN {X 0,Y 347.752,Z 155.164,A -85,B 0,C 180,E1 -13735.957,E2 -13735.957} C_VEL
LIN {X 0,Y 347.758,Z 155.217,A -85,B 0,C 180,E1 -13738.599,E2 -13738.599} C_VEL
LIN {X 0,Y 350.356,Z 166.477,A -85,B 0,C 180,E1 -13741.712,E2 -13741.712} C_VEL
LIN {X 0,Y 352.135,Z 175.806,A -85,B 0,C 180,E1 -13744.159,E2 -13744.159} C_VEL
LIN {X 0,Y 351.926,Z 180.185,A -85,B 0,C 180,E1 -13745.205,E2 -13745.205} C_VEL
LIN {X 0,Y 351.294,Z 186.162,A -85,B 0,C 180,E1 -13746.599,E2 -13746.599} C_VEL
LIN {X 0,Y 355.983,Z 212.379,A -85,B 0,C 180,E1 -13747.55,E2 -13747.55} C_VEL
LIN {X 0,Y 357.563,Z 224.655,A -85,B 0,C 180,E1 -13747.934,E2 -13747.934} C_VEL
LIN {X 0,Y 356.155,Z 295.266,A -85,B 0,C 180,E1 -13749.421,E2 -13749.421} C_VEL
LIN {X 0,Y 355.324,Z 309.079,A -85,B 0,C 180,E1 -13749.938,E2 -13749.938} C_VEL
LIN {X 0,Y 354.213,Z 322.04,A -85,B 0,C 180,E1 -13750.665,E2 -13750.665} C_VEL
LIN {X 0,Y 353.108,Z 333.83,A -85,B 0,C 180,E1 -13751.581,E2 -13751.581} C_VEL
LIN {X 0,Y 351.772,Z 345.209,A -85,B 0,C 180,E1 -13752.712,E2 -13752.712} C_VEL
LIN {X 0,Y 350.607,Z 355.192,A -85,B 0,C 180,E1 -13753.958,E2 -13753.958} C_VEL
LIN {X 0,Y 349.433,Z 364.743,A -85,B 0,C 180,E1 -13755.439,E2 -13755.439} C_VEL
LIN {X 0,Y 348.31,Z 373.757,A -85,B 0,C 180,E1 -13757.176,E2 -13757.176} C_VEL
LIN {X 0,Y 347.366,Z 381.03,A -85,B 0,C 180,E1 -13758.919,E2 -13758.919} C_VEL
LIN {X 0,Y 346.795,Z 386.855,A -85,B 0,C 180,E1 -13760.67,E2 -13760.67} C_VEL
LIN {X 0,Y 346.394,Z 391.452,A -85,B 0,C 180,E1 -13762.422,E2 -13762.422} C_VEL
LIN {X 0,Y 346.203,Z 394.959,A -85,B 0,C 180,E1 -13764.175,E2 -13764.175} C_VEL
LIN {X 0,Y 346.167,Z 396.717,A -85,B 0,C 180,E1 -13765.342,E2 -13765.342} C_VEL
LIN {X 0,Y 346.147,Z 398.063,A -85,B 0,C 180,E1 -13766.508,E2 -13766.508} C_VEL
LIN {X 0,Y 346.114,Z 399.013,A -85,B 0,C 180,E1 -13767.673,E2 -13767.673} C_VEL
LIN {X 0,Y 346.172,Z 399.562,A -85,B 0,C 180,E1 -13768.837,E2 -13768.837} C_VEL
LIN {X 0,Y 346.237,Z 399.675,A -85,B 0,C 180,E1 -13770,E2 -13770} C_VEL
LIN {X 0,Y 346.188,Z 399.392,A -85,B 0,C 180,E1 -13771.163,E2 -13771.163} C_VEL
LIN {X 0,Y 346.148,Z 397.642,A -85,B 0,C 180,E1 -13773.492,E2 -13773.492} C_VEL
LIN {X 0,Y 346.167,Z 396.106,A -85,B 0,C 180,E1 -13774.658,E2 -13774.658} C_VEL
LIN {X 0,Y 346.247,Z 393.006,A -85,B 0,C 180,E1 -13776.409,E2 -13776.409} C_VEL
LIN {X 0,Y 346.518,Z 388.834,A -85,B 0,C 180,E1 -13778.162,E2 -13778.162} C_VEL
LIN {X 0,Y 347.021,Z 382.455,A -85,B 0,C 180,E1 -13780.207,E2 -13780.207} C_VEL
LIN {X 0,Y 347.689,Z 375.503,A -85,B 0,C 180,E1 -13781.958,E2 -13781.958} C_VEL
LIN {X 0,Y 348.566,Z 368.405,A -85,B 0,C 180,E1 -13783.408,E2 -13783.408} C_VEL
LIN {X 0,Y 349.523,Z 359.824,A -85,B 0,C 180,E1 -13784.855,E2 -13784.855} C_VEL
LIN {X 0,Y 350.53,Z 349.213,A -85,B 0,C 180,E1 -13786.302,E2 -13786.302} C_VEL
LIN {X 0,Y 351.673,Z 338.719,A -85,B 0,C 180,E1 -13787.444,E2 -13787.444} C_VEL
LIN {X 0,Y 352.789,Z 327.167,A -85,B 0,C 180,E1 -13788.437,E2 -13788.437} C_VEL
LIN {X 0,Y 353.759,Z 315.192,A -85,B 0,C 180,E1 -13789.211,E2 -13789.211} C_VEL
LIN {X 0,Y 354.623,Z 301.371,A -85,B 0,C 180,E1 -13789.84,E2 -13789.84} C_VEL
LIN {X 0,Y 355.04,Z 288.646,A -85,B 0,C 180,E1 -13790.193,E2 -13790.193} C_VEL
LIN {X 0,Y 356.123,Z 222.477,A -85,B 0,C 180,E1 -13791.554,E2 -13791.554} C_VEL
LIN {X 0,Y 351.162,Z 190.648,A -85,B 0,C 180,E1 -13792.547,E2 -13792.547} C_VEL
LIN {X 0,Y 350.609,Z 186.927,A -85,B 0,C 180,E1 -13792.699,E2 -13792.699} C_VEL
LIN {X 0,Y 351.762,Z 175.382,A -85,B 0,C 180,E1 -13795.392,E2 -13795.392} C_VEL
LIN {X 0,Y 349.682,Z 164.027,A -85,B 0,C 180,E1 -13798.304,E2 -13798.304} C_VEL
LIN {X 0,Y 347.772,Z 155.169,A -85,B 0,C 180,E1 -13800.682,E2 -13800.682} C_VEL
LIN {X 0,Y 347.749,Z 155.165,A -85,B 0,C 180,E1 -13804.464,E2 -13804.464} C_VEL
LIN {X 0,Y 347.767,Z 155.164,A -85,B 0,C 180,E1 -13807.986,E2 -13807.986} C_VEL
LIN {X 0,Y 347.746,Z 155.167,A -85,B 0,C 180,E1 -13811.832,E2 -13811.832} C_VEL
LIN {X 0,Y 347.706,Z 155.173,A -85,B 0,C 180,E1 -13815.027,E2 -13815.027} C_VEL
LIN {X 0,Y 347.746,Z 155.165,A -85,B 0,C 180,E1 -13818.399,E2 -13818.399} C_VEL
LIN {X 0,Y 347.76,Z 155.165,A -85,B 0,C 180,E1 -13822.678,E2 -13822.678} C_VEL
LIN {X 0,Y 347.753,Z 155.164,A -85,B 0,C 180,E1 -13825.956,E2 -13825.956} C_VEL
LIN {X 0,Y 347.743,Z 155.166,A -85,B 0,C 180,E1 -13829.651,E2 -13829.651} C_VEL
LIN {X 0,Y 347.753,Z 155.164,A -85,B 0,C 180,E1 -13833.6,E2 -13833.6} C_VEL
LIN {X 0,Y 347.768,Z 155.163,A -85,B 0,C 180,E1 -13836.159,E2 -13836.159} C_VEL
LIN {X 0,Y 347.782,Z 155.161,A -85,B 0,C 180,E1 -13839.907,E2 -13839.907} C_VEL
LIN {X 0,Y 347.802,Z 155.158,A -85,B 0,C 180,E1 -13843.566,E2 -13843.566} C_VEL
LIN {X 0,Y 347.892,Z 155.148,A -85,B 0,C 180,E1 -13847.16,E2 -13847.16} C_VEL
LIN {X 0,Y 347.939,Z 155.144,A -85,B 0,C 180,E1 -13850.7,E2 -13850.7} C_VEL
LIN {X 0,Y 348.044,Z 155.132,A -85,B 0,C 180,E1 -13854.204,E2 -13854.204} C_VEL
LIN {X 0,Y 348.192,Z 155.11,A -85,B 0,C 180,E1 -13857.685,E2 -13857.685} C_VEL
LIN {X 0,Y 348.121,Z 155.118,A -85,B 0,C 180,E1 -13861.156,E2 -13861.156} C_VEL
LIN {X 0,Y 348.191,Z 155.114,A -85,B 0,C 180,E1 -13862.313,E2 -13862.313} C_VEL
LIN {X 0,Y 348.055,Z 155.126,A -85,B 0,C 180,E1 -13866.958,E2 -13866.958} C_VEL
LIN {X 0,Y 347.894,Z 155.148,A -85,B 0,C 180,E1 -13870.474,E2 -13870.474} C_VEL
LIN {X 0,Y 347.881,Z 155.152,A -85,B 0,C 180,E1 -13874.136,E2 -13874.136} C_VEL
LIN {X 0,Y 347.794,Z 155.161,A -85,B 0,C 180,E1 -13878.24,E2 -13878.24} C_VEL
LIN {X 0,Y 347.764,Z 155.168,A -85,B 0,C 180,E1 -13881.623,E2 -13881.623} C_VEL
LIN {X 0,Y 347.734,Z 155.168,A -85,B 0,C 180,E1 -13885.113,E2 -13885.113} C_VEL
LIN {X 0,Y 347.728,Z 155.172,A -85,B 0,C 180,E1 -13887.7,E2 -13887.7} C_VEL
LIN {X 0,Y 347.737,Z 155.166,A -85,B 0,C 180,E1 -13890.348,E2 -13890.348} C_VEL
LIN {X 0,Y 347.747,Z 155.166,A -85,B 0,C 180,E1 -13894.042,E2 -13894.042} C_VEL
LIN {X 0,Y 347.754,Z 155.17,A -85,B 0,C 180,E1 -13897.32,E2 -13897.32} C_VEL
LIN {X 0,Y 347.736,Z 155.169,A -85,B 0,C 180,E1 -13901.599,E2 -13901.599} C_VEL
LIN {X 0,Y 347.698,Z 155.176,A -85,B 0,C 180,E1 -13905.026,E2 -13905.026} C_VEL
LIN {X 0,Y 347.737,Z 155.167,A -85,B 0,C 180,E1 -13908.398,E2 -13908.398} C_VEL
LIN {X 0,Y 347.751,Z 155.168,A -85,B 0,C 180,E1 -13912.677,E2 -13912.677} C_VEL
LIN {X 0,Y 347.743,Z 155.165,A -85,B 0,C 180,E1 -13915.955,E2 -13915.955} C_VEL
LIN {X 0,Y 347.733,Z 155.167,A -85,B 0,C 180,E1 -13919.65,E2 -13919.65} C_VEL
LIN {X 0,Y 347.728,Z 155.167,A -85,B 0,C 180,E1 -13923.599,E2 -13923.599} C_VEL
LIN {X 0,Y 347.742,Z 155.167,A -85,B 0,C 180,E1 -13926.158,E2 -13926.158} C_VEL
LIN {X 0,Y 347.764,Z 155.163,A -85,B 0,C 180,E1 -13929.906,E2 -13929.906} C_VEL
LIN {X 0,Y 347.79,Z 155.16,A -85,B 0,C 180,E1 -13933.566,E2 -13933.566} C_VEL
LIN {X 0,Y 347.877,Z 155.149,A -85,B 0,C 180,E1 -13937.16,E2 -13937.16} C_VEL
LIN {X 0,Y 347.926,Z 155.145,A -85,B 0,C 180,E1 -13940.7,E2 -13940.7} C_VEL
LIN {X 0,Y 348.031,Z 155.136,A -85,B 0,C 180,E1 -13944.205,E2 -13944.205} C_VEL
LIN {X 0,Y 348.007,Z 155.25,A -85,B 0,C 180,E1 -13946.961,E2 -13946.961} C_VEL
LIN {X 0,Y 349.312,Z 161.756,A -85,B 0,C 180,E1 -13948.847,E2 -13948.847} C_VEL
LIN {X 0,Y 349.684,Z 163.478,A -85,B 0,C 180,E1 -13949.342,E2 -13949.342} C_VEL
LIN {X 0,Y 354.003,Z 176.651,A -85,B 0,C 180,E1 -13949.908,E2 -13949.908} C_VEL
LIN {X 0,Y 356.783,Z 191.197,A -85,B 0,C 180,E1 -13950.394,E2 -13950.394} C_VEL
LIN {X 0,Y 355.077,Z 271.339,A -85,B 0,C 180,E1 -13952.056,E2 -13952.056} C_VEL
LIN {X 0,Y 354.502,Z 284.435,A -85,B 0,C 180,E1 -13952.556,E2 -13952.556} C_VEL
LIN {X 0,Y 353.832,Z 297.028,A -85,B 0,C 180,E1 -13953.273,E2 -13953.273} C_VEL
LIN {X 0,Y 352.885,Z 309.516,A -85,B 0,C 180,E1 -13954.248,E2 -13954.248} C_VEL
LIN {X 0,Y 351.82,Z 321.33,A -85,B 0,C 180,E1 -13955.444,E2 -13955.444} C_VEL
LIN {X 0,Y 350.725,Z 331.609,A -85,B 0,C 180,E1 -13956.761,E2 -13956.761} C_VEL
LIN {X 0,Y 349.585,Z 341.702,A -85,B 0,C 180,E1 -13958.381,E2 -13958.381} C_VEL
LIN {X 0,Y 348.676,Z 349.204,A -85,B 0,C 180,E1 -13959.864,E2 -13959.864} C_VEL
LIN {X 0,Y 347.845,Z 356.549,A -85,B 0,C 180,E1 -13961.656,E2 -13961.656} C_VEL
LIN {X 0,Y 347.108,Z 362.839,A -85,B 0,C 180,E1 -13963.627,E2 -13963.627} C_VEL
LIN {X 0,Y 346.72,Z 366.941,A -85,B 0,C 180,E1 -13965.278,E2 -13965.278} C_VEL
LIN {X 0,Y 346.274,Z 370.925,A -85,B 0,C 180,E1 -13967.466,E2 -13967.466} C_VEL
LIN {X 0,Y 346.113,Z 372.742,A -85,B 0,C 180,E1 -13968.959,E2 -13968.959} C_VEL
LIN {X 0,Y 345.987,Z 374.105,A -85,B 0,C 180,E1 -13970.873,E2 -13970.873} C_VEL
LIN {X 0,Y 345.982,Z 374.405,A -85,B 0,C 180,E1 -13972.703,E2 -13972.703} C_VEL
LIN {X 0,Y 346.082,Z 374.05,A -85,B 0,C 180,E1 -13973.963,E2 -13973.963} C_VEL
LIN {X 0,Y 346.172,Z 373.22,A -85,B 0,C 180,E1 -13975.236,E2 -13975.236} C_VEL
LIN {X 0,Y 346.413,Z 371.533,A -85,B 0,C 180,E1 -13976.792,E2 -13976.792} C_VEL
LIN {X 0,Y 346.717,Z 368.909,A -85,B 0,C 180,E1 -13978.447,E2 -13978.447} C_VEL
LIN {X 0,Y 347.215,Z 364.664,A -85,B 0,C 180,E1 -13980.399,E2 -13980.399} C_VEL
LIN {X 0,Y 348.004,Z 358.744,A -85,B 0,C 180,E1 -13982.416,E2 -13982.416} C_VEL
LIN {X 0,Y 348.97,Z 351.421,A -85,B 0,C 180,E1 -13984.342,E2 -13984.342} C_VEL
LIN {X 0,Y 349.438,Z 348.123,A -85,B 0,C 180,E1 -13985.072,E2 -13985.072} C_VEL
LIN {X 0,Y 349.266,Z 344.516,A -85,B 0,C 180,E1 -13985.841,E2 -13985.841} C_VEL
LIN {X 0,Y 347.273,Z 338.398,A -85,B 0,C 180,E1 -13987.085,E2 -13987.085} C_VEL
LIN {X 0,Y 345.409,Z 331.827,A -85,B 0,C 180,E1 -13988.268,E2 -13988.268} C_VEL
LIN {X 0,Y 345.406,Z 327.383,A -85,B 0,C 180,E1 -13988.916,E2 -13988.916} C_VEL
LIN {X 0,Y 346.641,Z 316.913,A -85,B 0,C 180,E1 -13990.146,E2 -13990.146} C_VEL
LIN {X 0,Y 347.866,Z 305.158,A -85,B 0,C 180,E1 -13991.233,E2 -13991.233} C_VEL
LIN {X 0,Y 348.779,Z 293.502,A -85,B 0,C 180,E1 -13992.067,E2 -13992.067} C_VEL
LIN {X 0,Y 349.482,Z 280.944,A -85,B 0,C 180,E1 -13992.718,E2 -13992.718} C_VEL
LIN {X 0,Y 349.973,Z 268.611,A -85,B 0,C 180,E1 -13993.131,E2 -13993.131} C_VEL
LIN {X 0,Y 351.7,Z 191.42,A -85,B 0,C 180,E1 -13994.761,E2 -13994.761} C_VEL
LIN {X 0,Y 349.273,Z 180.691,A -85,B 0,C 180,E1 -13995.191,E2 -13995.191} C_VEL
LIN {X 0,Y 342.629,Z 164.292,A -85,B 0,C 180,E1 -13996.126,E2 -13996.126} C_VEL
LIN {X 0,Y 340.743,Z 156.041,A -85,B 0,C 180,E1 -13998.701,E2 -13998.701} C_VEL
LIN {X 0,Y 340.735,Z 156.047,A -85,B 0,C 180,E1 -14001.774,E2 -14001.774} C_VEL
LIN {X 0,Y 340.72,Z 156.047,A -85,B 0,C 180,E1 -14005.596,E2 -14005.596} C_VEL
LIN {X 0,Y 340.701,Z 156.045,A -85,B 0,C 180,E1 -14008.957,E2 -14008.957} C_VEL
LIN {X 0,Y 340.777,Z 156.036,A -85,B 0,C 180,E1 -14012.475,E2 -14012.475} C_VEL
LIN {X 0,Y 340.754,Z 156.038,A -85,B 0,C 180,E1 -14015.639,E2 -14015.639} C_VEL
LIN {X 0,Y 340.743,Z 156.039,A -85,B 0,C 180,E1 -14019.475,E2 -14019.475} C_VEL
LIN {X 0,Y 340.792,Z 156.032,A -85,B 0,C 180,E1 -14021.982,E2 -14021.982} C_VEL
LIN {X 0,Y 340.869,Z 156.021,A -85,B 0,C 180,E1 -14025.706,E2 -14025.706} C_VEL
LIN {X 0,Y 340.849,Z 156.026,A -85,B 0,C 180,E1 -14029.307,E2 -14029.307} C_VEL
LIN {X 0,Y 341.01,Z 156.008,A -85,B 0,C 180,E1 -14032.898,E2 -14032.898} C_VEL
LIN {X 0,Y 340.832,Z 156.018,A -85,B 0,C 180,E1 -14035.27,E2 -14035.27} C_VEL
LIN {X 0,Y 341.165,Z 155.982,A -85,B 0,C 180,E1 -14037.64,E2 -14037.64} C_VEL
LIN {X 0,Y 341.236,Z 155.97,A -85,B 0,C 180,E1 -14040.001,E2 -14040.001} C_VEL
LIN {X 0,Y 341.128,Z 155.986,A -85,B 0,C 180,E1 -14042.362,E2 -14042.362} C_VEL
LIN {X 0,Y 341.018,Z 155.993,A -85,B 0,C 180,E1 -14045.915,E2 -14045.915} C_VEL
LIN {X 0,Y 340.965,Z 156.012,A -85,B 0,C 180,E1 -14048.357,E2 -14048.357} C_VEL
LIN {X 0,Y 340.851,Z 156.016,A -85,B 0,C 180,E1 -14051.9,E2 -14051.9} C_VEL
LIN {X 0,Y 340.865,Z 156.023,A -85,B 0,C 180,E1 -14054.326,E2 -14054.326} C_VEL
LIN {X 0,Y 340.772,Z 156.036,A -85,B 0,C 180,E1 -14058.433,E2 -14058.433} C_VEL
LIN {X 0,Y 340.72,Z 156.035,A -85,B 0,C 180,E1 -14061.842,E2 -14061.842} C_VEL
LIN {X 0,Y 340.672,Z 156.042,A -85,B 0,C 180,E1 -14065.673,E2 -14065.673} C_VEL
LIN {X 0,Y 340.681,Z 156.047,A -85,B 0,C 180,E1 -14068.326,E2 -14068.326} C_VEL
LIN {X 0,Y 340.694,Z 156.039,A -85,B 0,C 180,E1 -14071.046,E2 -14071.046} C_VEL
LIN {X 0,Y 340.717,Z 156.04,A -85,B 0,C 180,E1 -14075.28,E2 -14075.28} C_VEL
LIN {X 0,Y 340.695,Z 156.041,A -85,B 0,C 180,E1 -14078.383,E2 -14078.383} C_VEL
LIN {X 0,Y 340.693,Z 156.048,A -85,B 0,C 180,E1 -14082.044,E2 -14082.044} C_VEL
LIN {X 0,Y 340.652,Z 156.057,A -85,B 0,C 180,E1 -14086.228,E2 -14086.228} C_VEL
LIN {X 0,Y 340.67,Z 156.053,A -85,B 0,C 180,E1 -14088.688,E2 -14088.688} C_VEL
LIN {X 0,Y 340.721,Z 156.044,A -85,B 0,C 180,E1 -14091.771,E2 -14091.771} C_VEL
LIN {X 0,Y 340.726,Z 156.04,A -85,B 0,C 180,E1 -14095.596,E2 -14095.596} C_VEL
LIN {X 0,Y 340.723,Z 156.142,A -85,B 0,C 180,E1 -14098.139,E2 -14098.139} C_VEL
LIN {X 0,Y 343.222,Z 166.822,A -85,B 0,C 180,E1 -14101.179,E2 -14101.179} C_VEL
LIN {X 0,Y 345.04,Z 176.037,A -85,B 0,C 180,E1 -14103.667,E2 -14103.667} C_VEL
LIN {X 0,Y 345.314,Z 178.996,A -85,B 0,C 180,E1 -14104.426,E2 -14104.426} C_VEL
LIN {X 0,Y 344.525,Z 185.925,A -85,B 0,C 180,E1 -14106.078,E2 -14106.078} C_VEL
LIN {X 0,Y 349.188,Z 211.48,A -85,B 0,C 180,E1 -14107.034,E2 -14107.034} C_VEL
LIN {X 0,Y 351.067,Z 224.986,A -85,B 0,C 180,E1 -14107.479,E2 -14107.479} C_VEL
LIN {X 0,Y 349.594,Z 294.945,A -85,B 0,C 180,E1 -14108.979,E2 -14108.979} C_VEL
LIN {X 0,Y 348.736,Z 308.762,A -85,B 0,C 180,E1 -14109.503,E2 -14109.503} C_VEL
LIN {X 0,Y 347.657,Z 321.203,A -85,B 0,C 180,E1 -14110.208,E2 -14110.208} C_VEL
LIN {X 0,Y 346.588,Z 332.327,A -85,B 0,C 180,E1 -14111.068,E2 -14111.068} C_VEL
LIN {X 0,Y 345.187,Z 343.92,A -85,B 0,C 180,E1 -14112.218,E2 -14112.218} C_VEL
LIN {X 0,Y 343.824,Z 354.322,A -85,B 0,C 180,E1 -14113.516,E2 -14113.516} C_VEL
LIN {X 0,Y 342.804,Z 362.943,A -85,B 0,C 180,E1 -14114.847,E2 -14114.847} C_VEL
LIN {X 0,Y 341.777,Z 370.867,A -85,B 0,C 180,E1 -14116.322,E2 -14116.322} C_VEL
LIN {X 0,Y 340.611,Z 378.617,A -85,B 0,C 180,E1 -14118.093,E2 -14118.093} C_VEL
LIN {X 0,Y 339.945,Z 384.858,A -85,B 0,C 180,E1 -14119.879,E2 -14119.879} C_VEL
LIN {X 0,Y 339.462,Z 389.828,A -85,B 0,C 180,E1 -14121.667,E2 -14121.667} C_VEL
LIN {X 0,Y 339.163,Z 393.671,A -85,B 0,C 180,E1 -14123.456,E2 -14123.456} C_VEL
LIN {X 0,Y 339.069,Z 396.491,A -85,B 0,C 180,E1 -14125.244,E2 -14125.244} C_VEL
LIN {X 0,Y 339.071,Z 397.831,A -85,B 0,C 180,E1 -14126.435,E2 -14126.435} C_VEL
LIN {X 0,Y 339.026,Z 398.773,A -85,B 0,C 180,E1 -14127.624,E2 -14127.624} C_VEL
LIN {X 0,Y 339.073,Z 399.308,A -85,B 0,C 180,E1 -14128.813,E2 -14128.813} C_VEL
LIN {X 0,Y 339.141,Z 399.411,A -85,B 0,C 180,E1 -14130,E2 -14130} C_VEL
LIN {X 0,Y 339.088,Z 399.119,A -85,B 0,C 180,E1 -14131.188,E2 -14131.188} C_VEL
LIN {X 0,Y 339.028,Z 398.437,A -85,B 0,C 180,E1 -14132.376,E2 -14132.376} C_VEL
LIN {X 0,Y 339.072,Z 397.347,A -85,B 0,C 180,E1 -14133.565,E2 -14133.565} C_VEL
LIN {X 0,Y 339.114,Z 394.005,A -85,B 0,C 180,E1 -14135.851,E2 -14135.851} C_VEL
LIN {X 0,Y 339.346,Z 390.004,A -85,B 0,C 180,E1 -14137.737,E2 -14137.737} C_VEL
LIN {X 0,Y 339.727,Z 385.039,A -85,B 0,C 180,E1 -14139.526,E2 -14139.526} C_VEL
LIN {X 0,Y 340.282,Z 378.783,A -85,B 0,C 180,E1 -14141.316,E2 -14141.316} C_VEL
LIN {X 0,Y 341.268,Z 370.979,A -85,B 0,C 180,E1 -14143.093,E2 -14143.093} C_VEL
LIN {X 0,Y 342.36,Z 361.457,A -85,B 0,C 180,E1 -14144.824,E2 -14144.824} C_VEL
LIN {X 0,Y 343.424,Z 351.281,A -85,B 0,C 180,E1 -14146.313,E2 -14146.313} C_VEL
LIN {X 0,Y 344.543,Z 341.004,A -85,B 0,C 180,E1 -14147.51,E2 -14147.51} C_VEL
LIN {X 0,Y 345.67,Z 330.084,A -85,B 0,C 180,E1 -14148.523,E2 -14148.523} C_VEL
LIN {X 0,Y 346.745,Z 318.039,A -85,B 0,C 180,E1 -14149.384,E2 -14149.384} C_VEL
LIN {X 0,Y 347.713,Z 304.855,A -85,B 0,C 180,E1 -14150.059,E2 -14150.059} C_VEL
LIN {X 0,Y 348.287,Z 291.683,A -85,B 0,C 180,E1 -14150.486,E2 -14150.486} C_VEL
LIN {X 0,Y 349.417,Z 223.106,A -85,B 0,C 180,E1 -14151.936,E2 -14151.936} C_VEL
LIN {X 0,Y 344.455,Z 191.147,A -85,B 0,C 180,E1 -14152.959,E2 -14152.959} C_VEL
LIN {X 0,Y 343.791,Z 186.71,A -85,B 0,C 180,E1 -14153.129,E2 -14153.129} C_VEL
LIN {X 0,Y 344.794,Z 177.388,A -85,B 0,C 180,E1 -14155.344,E2 -14155.344} C_VEL
LIN {X 0,Y 343.577,Z 169.412,A -85,B 0,C 180,E1 -14157.403,E2 -14157.403} C_VEL
LIN {X 0,Y 340.931,Z 156.984,A -85,B 0,C 180,E1 -14160.77,E2 -14160.77} C_VEL
LIN {X 0,Y 340.739,Z 156.044,A -85,B 0,C 180,E1 -14161.041,E2 -14161.041} C_VEL
LIN {X 0,Y 340.722,Z 156.044,A -85,B 0,C 180,E1 -14165.279,E2 -14165.279} C_VEL
LIN {X 0,Y 340.698,Z 156.043,A -85,B 0,C 180,E1 -14168.382,E2 -14168.382} C_VEL
LIN {X 0,Y 340.696,Z 156.043,A -85,B 0,C 180,E1 -14172.044,E2 -14172.044} C_VEL
LIN {X 0,Y 340.655,Z 156.048,A -85,B 0,C 180,E1 -14176.227,E2 -14176.227} C_VEL
LIN {X 0,Y 340.676,Z 156.047,A -85,B 0,C 180,E1 -14178.688,E2 -14178.688} C_VEL
LIN {X 0,Y 340.724,Z 156.041,A -85,B 0,C 180,E1 -14181.77,E2 -14181.77} C_VEL
LIN {X 0,Y 340.727,Z 156.041,A -85,B 0,C 180,E1 -14185.595,E2 -14185.595} C_VEL
LIN {X 0,Y 340.698,Z 156.049,A -85,B 0,C 180,E1 -14188.954,E2 -14188.954} C_VEL
LIN {X 0,Y 340.724,Z 156.044,A -85,B 0,C 180,E1 -14193.012,E2 -14193.012} C_VEL
LIN {X 0,Y 340.744,Z 156.037,A -85,B 0,C 180,E1 -14195.637,E2 -14195.637} C_VEL
LIN {X 0,Y 340.719,Z 156.041,A -85,B 0,C 180,E1 -14199.472,E2 -14199.472} C_VEL
LIN {X 0,Y 340.765,Z 156.035,A -85,B 0,C 180,E1 -14201.978,E2 -14201.978} C_VEL
LIN {X 0,Y 340.837,Z 156.026,A -85,B 0,C 180,E1 -14205.729,E2 -14205.729} C_VEL
LIN {X 0,Y 340.852,Z 156.024,A -85,B 0,C 180,E1 -14209.305,E2 -14209.305} C_VEL
LIN {X 0,Y 341.006,Z 156.005,A -85,B 0,C 180,E1 -14212.896,E2 -14212.896} C_VEL
LIN {X 0,Y 340.816,Z 156.028,A -85,B 0,C 180,E1 -14215.268,E2 -14215.268} C_VEL
LIN {X 0,Y 341.129,Z 155.99,A -85,B 0,C 180,E1 -14217.638,E2 -14217.638} C_VEL
LIN {X 0,Y 341.093,Z 155.993,A -85,B 0,C 180,E1 -14221.18,E2 -14221.18} C_VEL
LIN {X 0,Y 341.128,Z 155.992,A -85,B 0,C 180,E1 -14222.361,E2 -14222.361} C_VEL
LIN {X 0,Y 340.991,Z 156.006,A -85,B 0,C 180,E1 -14226.484,E2 -14226.484} C_VEL
LIN {X 0,Y 340.883,Z 156.021,A -85,B 0,C 180,E1 -14229.493,E2 -14229.493} C_VEL
LIN {X 0,Y 340.843,Z 156.025,A -85,B 0,C 180,E1 -14233.109,E2 -14233.109} C_VEL
LIN {X 0,Y 340.734,Z 156.037,A -85,B 0,C 180,E1 -14236.783,E2 -14236.783} C_VEL
LIN {X 0,Y 340.7,Z 156.044,A -85,B 0,C 180,E1 -14239.271,E2 -14239.271} C_VEL
LIN {X 0,Y 340.7,Z 156.044,A -85,B 0,C 180,E1 -14243.074,E2 -14243.074} C_VEL
LIN {X 0,Y 340.709,Z 156.042,A -85,B 0,C 180,E1 -14246.987,E2 -14246.987} C_VEL
LIN {X 0,Y 340.692,Z 156.045,A -85,B 0,C 180,E1 -14251.044,E2 -14251.044} C_VEL
LIN {X 0,Y 340.716,Z 156.046,A -85,B 0,C 180,E1 -14255.278,E2 -14255.278} C_VEL
LIN {X 0,Y 340.691,Z 156.043,A -85,B 0,C 180,E1 -14258.381,E2 -14258.381} C_VEL
LIN {X 0,Y 340.689,Z 156.044,A -85,B 0,C 180,E1 -14262.043,E2 -14262.043} C_VEL
LIN {X 0,Y 340.646,Z 156.049,A -85,B 0,C 180,E1 -14266.226,E2 -14266.226} C_VEL
LIN {X 0,Y 340.667,Z 156.049,A -85,B 0,C 180,E1 -14268.687,E2 -14268.687} C_VEL
LIN {X 0,Y 340.714,Z 156.041,A -85,B 0,C 180,E1 -14271.77,E2 -14271.77} C_VEL
LIN {X 0,Y 340.717,Z 156.041,A -85,B 0,C 180,E1 -14275.595,E2 -14275.595} C_VEL
LIN {X 0,Y 340.688,Z 156.049,A -85,B 0,C 180,E1 -14278.954,E2 -14278.954} C_VEL
LIN {X 0,Y 340.704,Z 156.045,A -85,B 0,C 180,E1 -14283.011,E2 -14283.011} C_VEL
LIN {X 0,Y 340.694,Z 156.046,A -85,B 0,C 180,E1 -14286.924,E2 -14286.924} C_VEL
LIN {X 0,Y 340.697,Z 156.047,A -85,B 0,C 180,E1 -14290.728,E2 -14290.728} C_VEL
LIN {X 0,Y 340.786,Z 156.038,A -85,B 0,C 180,E1 -14294.449,E2 -14294.449} C_VEL
LIN {X 0,Y 340.838,Z 156.029,A -85,B 0,C 180,E1 -14298.1,E2 -14298.1} C_VEL
LIN {X 0,Y 340.973,Z 156.01,A -85,B 0,C 180,E1 -14301.704,E2 -14301.704} C_VEL
LIN {X 0,Y 341.006,Z 156.01,A -85,B 0,C 180,E1 -14304.085,E2 -14304.085} C_VEL
LIN {X 0,Y 340.885,Z 156.045,A -85,B 0,C 180,E1 -14306.602,E2 -14306.602} C_VEL
LIN {X 0,Y 342.319,Z 162.537,A -85,B 0,C 180,E1 -14308.529,E2 -14308.529} C_VEL
LIN {X 0,Y 342.505,Z 163.738,A -85,B 0,C 180,E1 -14308.877,E2 -14308.877} C_VEL
LIN {X 0,Y 347.561,Z 178.653,A -85,B 0,C 180,E1 -14309.546,E2 -14309.546} C_VEL
LIN {X 0,Y 350.128,Z 191.737,A -85,B 0,C 180,E1 -14310,E2 -14310} C_VEL
LIN {X 0,Y 348.409,Z 270.753,A -85,B 0,C 180,E1 -14311.661,E2 -14311.661} C_VEL
LIN {X 0,Y 347.86,Z 283.348,A -85,B 0,C 180,E1 -14312.135,E2 -14312.135} C_VEL
LIN {X 0,Y 347.098,Z 296.88,A -85,B 0,C 180,E1 -14312.901,E2 -14312.901} C_VEL
LIN {X 0,Y 346.148,Z 309.168,A -85,B 0,C 180,E1 -14313.865,E2 -14313.865} C_VEL
LIN {X 0,Y 345.124,Z 320.044,A -85,B 0,C 180,E1 -14314.965,E2 -14314.965} C_VEL
LIN {X 0,Y 343.993,Z 330.642,A -85,B 0,C 180,E1 -14316.304,E2 -14316.304} C_VEL
LIN {X 0,Y 342.999,Z 339.289,A -85,B 0,C 180,E1 -14317.653,E2 -14317.653} C_VEL
LIN {X 0,Y 341.862,Z 348.034,A -85,B 0,C 180,E1 -14319.334,E2 -14319.334} C_VEL
LIN {X 0,Y 340.903,Z 356.153,A -85,B 0,C 180,E1 -14321.294,E2 -14321.294} C_VEL
LIN {X 0,Y 340.188,Z 362.144,A -85,B 0,C 180,E1 -14323.135,E2 -14323.135} C_VEL
LIN {X 0,Y 339.705,Z 366.818,A -85,B 0,C 180,E1 -14324.987,E2 -14324.987} C_VEL
LIN {X 0,Y 339.297,Z 370.359,A -85,B 0,C 180,E1 -14326.857,E2 -14326.857} C_VEL
LIN {X 0,Y 339.12,Z 372.108,A -85,B 0,C 180,E1 -14328.111,E2 -14328.111} C_VEL
LIN {X 0,Y 338.97,Z 373.431,A -85,B 0,C 180,E1 -14329.374,E2 -14329.374} C_VEL
LIN {X 0,Y 338.888,Z 374.44,A -85,B 0,C 180,E1 -14331.06,E2 -14331.06} C_VEL
LIN {X 0,Y 338.936,Z 374.61,A -85,B 0,C 180,E1 -14333.202,E2 -14333.202} C_VEL
LIN {X 0,Y 339.024,Z 374.066,A -85,B 0,C 180,E1 -14334.494,E2 -14334.494} C_VEL
LIN {X 0,Y 339.139,Z 373.051,A -85,B 0,C 180,E1 -14335.797,E2 -14335.797} C_VEL
LIN {X 0,Y 339.513,Z 370.6,A -85,B 0,C 180,E1 -14337.759,E2 -14337.759} C_VEL
LIN {X 0,Y 339.927,Z 366.923,A -85,B 0,C 180,E1 -14339.749,E2 -14339.749} C_VEL
LIN {X 0,Y 340.604,Z 362.034,A -85,B 0,C 180,E1 -14341.683,E2 -14341.683} C_VEL
LIN {X 0,Y 341.56,Z 355.166,A -85,B 0,C 180,E1 -14343.749,E2 -14343.749} C_VEL
LIN {X 0,Y 342.594,Z 348.169,A -85,B 0,C 180,E1 -14345.417,E2 -14345.417} C_VEL
LIN {X 0,Y 343.838,Z 339.181,A -85,B 0,C 180,E1 -14347.143,E2 -14347.143} C_VEL
LIN {X 0,Y 345.071,Z 329.778,A -85,B 0,C 180,E1 -14348.589,E2 -14348.589} C_VEL
LIN {X 0,Y 345.406,Z 327.383,A -85,B 0,C 180,E1 -14348.916,E2 -14348.916} C_VEL
LIN {X 0,Y 345.437,Z 322.827,A -85,B 0,C 180,E1 -14349.539,E2 -14349.539} C_VEL
LIN {X 0,Y 343.681,Z 315.224,A -85,B 0,C 180,E1 -14350.556,E2 -14350.556} C_VEL
LIN {X 0,Y 341.777,Z 307.192,A -85,B 0,C 180,E1 -14351.474,E2 -14351.474} C_VEL
LIN {X 0,Y 341.564,Z 301.962,A -85,B 0,C 180,E1 -14351.933,E2 -14351.933} C_VEL
LIN {X 0,Y 342.422,Z 289.924,A -85,B 0,C 180,E1 -14352.733,E2 -14352.733} C_VEL
LIN {X 0,Y 343.105,Z 277.257,A -85,B 0,C 180,E1 -14353.33,E2 -14353.33} C_VEL
LIN {X 0,Y 343.605,Z 263.79,A -85,B 0,C 180,E1 -14353.706,E2 -14353.706} C_VEL
LIN {X 0,Y 345.17,Z 192.134,A -85,B 0,C 180,E1 -14355.246,E2 -14355.246} C_VEL
LIN {X 0,Y 343.142,Z 183.243,A -85,B 0,C 180,E1 -14355.616,E2 -14355.616} C_VEL
LIN {X 0,Y 336.373,Z 166.912,A -85,B 0,C 180,E1 -14356.573,E2 -14356.573} C_VEL
LIN {X 0,Y 335.494,Z 164.49,A -85,B 0,C 180,E1 -14356.753,E2 -14356.753} C_VEL
LIN {X 0,Y 333.718,Z 156.92,A -85,B 0,C 180,E1 -14359.195,E2 -14359.195} C_VEL
LIN {X 0,Y 333.663,Z 156.928,A -85,B 0,C 180,E1 -14363.168,E2 -14363.168} C_VEL
LIN {X 0,Y 333.671,Z 156.926,A -85,B 0,C 180,E1 -14365.342,E2 -14365.342} C_VEL
LIN {X 0,Y 333.7,Z 156.917,A -85,B 0,C 180,E1 -14369.711,E2 -14369.711} C_VEL
LIN {X 0,Y 333.741,Z 156.912,A -85,B 0,C 180,E1 -14372.402,E2 -14372.402} C_VEL
LIN {X 0,Y 333.726,Z 156.916,A -85,B 0,C 180,E1 -14375.092,E2 -14375.092} C_VEL
LIN {X 0,Y 333.678,Z 156.918,A -85,B 0,C 180,E1 -14379.02,E2 -14379.02} C_VEL
LIN {X 0,Y 333.74,Z 156.911,A -85,B 0,C 180,E1 -14381.588,E2 -14381.588} C_VEL
LIN {X 0,Y 333.808,Z 156.901,A -85,B 0,C 180,E1 -14385.578,E2 -14385.578} C_VEL
LIN {X 0,Y 333.818,Z 156.903,A -85,B 0,C 180,E1 -14389.079,E2 -14389.079} C_VEL
LIN {X 0,Y 333.963,Z 156.883,A -85,B 0,C 180,E1 -14392.747,E2 -14392.747} C_VEL
LIN {X 0,Y 333.797,Z 156.895,A -85,B 0,C 180,E1 -14395.17,E2 -14395.17} C_VEL
LIN {X 0,Y 334.102,Z 156.862,A -85,B 0,C 180,E1 -14397.59,E2 -14397.59} C_VEL
LIN {X 0,Y 334.189,Z 156.847,A -85,B 0,C 180,E1 -14400.001,E2 -14400.001} C_VEL
LIN {X 0,Y 334.069,Z 156.866,A -85,B 0,C 180,E1 -14402.412,E2 -14402.412} C_VEL
LIN {X 0,Y 333.992,Z 156.868,A -85,B 0,C 180,E1 -14406.04,E2 -14406.04} C_VEL
LIN {X 0,Y 333.822,Z 156.898,A -85,B 0,C 180,E1 -14409.697,E2 -14409.697} C_VEL
LIN {X 0,Y 333.794,Z 156.904,A -85,B 0,C 180,E1 -14413.392,E2 -14413.392} C_VEL
LIN {X 0,Y 333.726,Z 156.905,A -85,B 0,C 180,E1 -14415.89,E2 -14415.89} C_VEL
LIN {X 0,Y 333.71,Z 156.915,A -85,B 0,C 180,E1 -14418.61,E2 -14418.61} C_VEL
LIN {X 0,Y 333.651,Z 156.918,A -85,B 0,C 180,E1 -14422.282,E2 -14422.282} C_VEL
LIN {X 0,Y 333.66,Z 156.921,A -85,B 0,C 180,E1 -14425.079,E2 -14425.079} C_VEL
LIN {X 0,Y 333.652,Z 156.924,A -85,B 0,C 180,E1 -14428.979,E2 -14428.979} C_VEL
LIN {X 0,Y 333.646,Z 156.924,A -85,B 0,C 180,E1 -14432.587,E2 -14432.587} C_VEL
LIN {X 0,Y 333.675,Z 156.92,A -85,B 0,C 180,E1 -14436.14,E2 -14436.14} C_VEL
LIN {X 0,Y 333.622,Z 156.929,A -85,B 0,C 180,E1 -14439.197,E2 -14439.197} C_VEL
LIN {X 0,Y 333.628,Z 156.93,A -85,B 0,C 180,E1 -14442.499,E2 -14442.499} C_VEL
LIN {X 0,Y 333.596,Z 156.935,A -85,B 0,C 180,E1 -14445.955,E2 -14445.955} C_VEL
LIN {X 0,Y 333.604,Z 156.933,A -85,B 0,C 180,E1 -14449.325,E2 -14449.325} C_VEL
LIN {X 0,Y 333.665,Z 156.915,A -85,B 0,C 180,E1 -14453.169,E2 -14453.169} C_VEL
LIN {X 0,Y 333.677,Z 156.92,A -85,B 0,C 180,E1 -14455.342,E2 -14455.342} C_VEL
LIN {X 0,Y 333.682,Z 157.004,A -85,B 0,C 180,E1 -14457.633,E2 -14457.633} C_VEL
LIN {X 0,Y 336.039,Z 166.974,A -85,B 0,C 180,E1 -14460.563,E2 -14460.563} C_VEL
LIN {X 0,Y 338.229,Z 177.895,A -85,B 0,C 180,E1 -14463.591,E2 -14463.591} C_VEL
LIN {X 0,Y 338.326,Z 181.309,A -85,B 0,C 180,E1 -14464.467,E2 -14464.467} C_VEL
LIN {X 0,Y 337.792,Z 185.652,A -85,B 0,C 180,E1 -14465.523,E2 -14465.523} C_VEL
LIN {X 0,Y 342.667,Z 212.057,A -85,B 0,C 180,E1 -14466.549,E2 -14466.549} C_VEL
LIN {X 0,Y 344.577,Z 226.034,A -85,B 0,C 180,E1 -14467.022,E2 -14467.022} C_VEL
LIN {X 0,Y 343.056,Z 294.624,A -85,B 0,C 180,E1 -14468.519,E2 -14468.519} C_VEL
LIN {X 0,Y 342.164,Z 308.455,A -85,B 0,C 180,E1 -14469.052,E2 -14469.052} C_VEL
LIN {X 0,Y 341.006,Z 321.43,A -85,B 0,C 180,E1 -14469.805,E2 -14469.805} C_VEL
LIN {X 0,Y 339.884,Z 332.433,A -85,B 0,C 180,E1 -14470.68,E2 -14470.68} C_VEL
LIN {X 0,Y 338.433,Z 343.959,A -85,B 0,C 180,E1 -14471.851,E2 -14471.851} C_VEL
LIN {X 0,Y 336.972,Z 354.472,A -85,B 0,C 180,E1 -14473.195,E2 -14473.195} C_VEL
LIN {X 0,Y 335.948,Z 362.889,A -85,B 0,C 180,E1 -14474.53,E2 -14474.53} C_VEL
LIN {X 0,Y 334.864,Z 370.767,A -85,B 0,C 180,E1 -14476.034,E2 -14476.034} C_VEL
LIN {X 0,Y 333.645,Z 378.473,A -85,B 0,C 180,E1 -14477.84,E2 -14477.84} C_VEL
LIN {X 0,Y 332.915,Z 384.687,A -85,B 0,C 180,E1 -14479.663,E2 -14479.663} C_VEL
LIN {X 0,Y 332.417,Z 389.636,A -85,B 0,C 180,E1 -14481.489,E2 -14481.489} C_VEL
LIN {X 0,Y 332.099,Z 393.462,A -85,B 0,C 180,E1 -14483.316,E2 -14483.316} C_VEL
LIN {X 0,Y 331.976,Z 396.266,A -85,B 0,C 180,E1 -14485.143,E2 -14485.143} C_VEL
LIN {X 0,Y 331.996,Z 397.599,A -85,B 0,C 180,E1 -14486.359,E2 -14486.359} C_VEL
LIN {X 0,Y 331.941,Z 398.533,A -85,B 0,C 180,E1 -14487.573,E2 -14487.573} C_VEL
LIN {X 0,Y 331.975,Z 399.052,A -85,B 0,C 180,E1 -14488.787,E2 -14488.787} C_VEL
LIN {X 0,Y 332.045,Z 399.147,A -85,B 0,C 180,E1 -14490,E2 -14490} C_VEL
LIN {X 0,Y 331.989,Z 398.847,A -85,B 0,C 180,E1 -14491.213,E2 -14491.213} C_VEL
LIN {X 0,Y 331.943,Z 398.157,A -85,B 0,C 180,E1 -14492.427,E2 -14492.427} C_VEL
LIN {X 0,Y 331.997,Z 397.052,A -85,B 0,C 180,E1 -14493.641,E2 -14493.641} C_VEL
LIN {X 0,Y 332.01,Z 394.028,A -85,B 0,C 180,E1 -14495.784,E2 -14495.784} C_VEL
LIN {X 0,Y 332.271,Z 389.667,A -85,B 0,C 180,E1 -14497.903,E2 -14497.903} C_VEL
LIN {X 0,Y 332.7,Z 384.682,A -85,B 0,C 180,E1 -14499.73,E2 -14499.73} C_VEL
LIN {X 0,Y 333.292,Z 378.403,A -85,B 0,C 180,E1 -14501.556,E2 -14501.556} C_VEL
LIN {X 0,Y 334.32,Z 370.556,A -85,B 0,C 180,E1 -14503.37,E2 -14503.37} C_VEL
LIN {X 0,Y 335.416,Z 361.41,A -85,B 0,C 180,E1 -14505.067,E2 -14505.067} C_VEL
LIN {X 0,Y 336.477,Z 351.656,A -85,B 0,C 180,E1 -14506.534,E2 -14506.534} C_VEL
LIN {X 0,Y 337.773,Z 340.43,A -85,B 0,C 180,E1 -14507.873,E2 -14507.873} C_VEL
LIN {X 0,Y 338.941,Z 329.434,A -85,B 0,C 180,E1 -14508.905,E2 -14508.905} C_VEL
LIN {X 0,Y 340.054,Z 317.28,A -85,B 0,C 180,E1 -14509.781,E2 -14509.781} C_VEL
LIN {X 0,Y 340.985,Z 304.696,A -85,B 0,C 180,E1 -14510.432,E2 -14510.432} C_VEL
LIN {X 0,Y 341.578,Z 291.591,A -85,B 0,C 180,E1 -14510.868,E2 -14510.868} C_VEL
LIN {X 0,Y 342.863,Z 224.589,A -85,B 0,C 180,E1 -14512.305,E2 -14512.305} C_VEL
LIN {X 0,Y 337.527,Z 190.096,A -85,B 0,C 180,E1 -14513.435,E2 -14513.435} C_VEL
LIN {X 0,Y 336.982,Z 186.505,A -85,B 0,C 180,E1 -14513.572,E2 -14513.572} C_VEL
LIN {X 0,Y 337.836,Z 178.278,A -85,B 0,C 180,E1 -14515.574,E2 -14515.574} C_VEL
LIN {X 0,Y 336.565,Z 170.38,A -85,B 0,C 180,E1 -14517.661,E2 -14517.661} C_VEL
LIN {X 0,Y 333.974,Z 158.209,A -85,B 0,C 180,E1 -14521.035,E2 -14521.035} C_VEL
LIN {X 0,Y 333.671,Z 156.923,A -85,B 0,C 180,E1 -14521.42,E2 -14521.42} C_VEL
LIN {X 0,Y 333.69,Z 156.917,A -85,B 0,C 180,E1 -14524.774,E2 -14524.774} C_VEL
LIN {X 0,Y 333.648,Z 156.925,A -85,B 0,C 180,E1 -14527.652,E2 -14527.652} C_VEL
LIN {X 0,Y 333.608,Z 156.928,A -85,B 0,C 180,E1 -14530.774,E2 -14530.774} C_VEL
LIN {X 0,Y 333.595,Z 156.928,A -85,B 0,C 180,E1 -14534.25,E2 -14534.25} C_VEL
LIN {X 0,Y 333.642,Z 156.925,A -85,B 0,C 180,E1 -14537.617,E2 -14537.617} C_VEL
LIN {X 0,Y 333.639,Z 156.928,A -85,B 0,C 180,E1 -14541.206,E2 -14541.206} C_VEL
LIN {X 0,Y 333.678,Z 156.918,A -85,B 0,C 180,E1 -14543.86,E2 -14543.86} C_VEL
LIN {X 0,Y 333.649,Z 156.924,A -85,B 0,C 180,E1 -14547.413,E2 -14547.413} C_VEL
LIN {X 0,Y 333.658,Z 156.925,A -85,B 0,C 180,E1 -14551.022,E2 -14551.022} C_VEL
LIN {X 0,Y 333.701,Z 156.918,A -85,B 0,C 180,E1 -14555.088,E2 -14555.088} C_VEL
LIN {X 0,Y 333.659,Z 156.923,A -85,B 0,C 180,E1 -14559.017,E2 -14559.017} C_VEL
LIN {X 0,Y 333.717,Z 156.913,A -85,B 0,C 180,E1 -14561.584,E2 -14561.584} C_VEL
LIN {X 0,Y 333.778,Z 156.905,A -85,B 0,C 180,E1 -14565.599,E2 -14565.599} C_VEL
LIN {X 0,Y 333.821,Z 156.9,A -85,B 0,C 180,E1 -14569.077,E2 -14569.077} C_VEL
LIN {X 0,Y 333.961,Z 156.883,A -85,B 0,C 180,E1 -14572.745,E2 -14572.745} C_VEL
LIN {X 0,Y 333.782,Z 156.904,A -85,B 0,C 180,E1 -14575.168,E2 -14575.168} C_VEL
LIN {X 0,Y 334.07,Z 156.869,A -85,B 0,C 180,E1 -14577.588,E2 -14577.588} C_VEL
LIN {X 0,Y 334.063,Z 156.868,A -85,B 0,C 180,E1 -14581.204,E2 -14581.204} C_VEL
LIN {X 0,Y 334.068,Z 156.87,A -85,B 0,C 180,E1 -14582.41,E2 -14582.41} C_VEL
LIN {X 0,Y 333.96,Z 156.883,A -85,B 0,C 180,E1 -14586.475,E2 -14586.475} C_VEL
LIN {X 0,Y 333.821,Z 156.903,A -85,B 0,C 180,E1 -14589.695,E2 -14589.695} C_VEL
LIN {X 0,Y 333.788,Z 156.904,A -85,B 0,C 180,E1 -14593.391,E2 -14593.391} C_VEL
LIN {X 0,Y 333.68,Z 156.916,A -85,B 0,C 180,E1 -14597.149,E2 -14597.149} C_VEL
LIN {X 0,Y 333.645,Z 156.926,A -85,B 0,C 180,E1 -14599.695,E2 -14599.695} C_VEL
LIN {X 0,Y 333.649,Z 156.922,A -85,B 0,C 180,E1 -14602.28,E2 -14602.28} C_VEL
LIN {X 0,Y 333.656,Z 156.921,A -85,B 0,C 180,E1 -14605.076,E2 -14605.076} C_VEL
LIN {X 0,Y 333.63,Z 156.923,A -85,B 0,C 180,E1 -14608.978,E2 -14608.978} C_VEL
LIN {X 0,Y 333.642,Z 156.922,A -85,B 0,C 180,E1 -14612.586,E2 -14612.586} C_VEL
LIN {X 0,Y 333.673,Z 156.917,A -85,B 0,C 180,E1 -14616.138,E2 -14616.138} C_VEL
LIN {X 0,Y 333.617,Z 156.928,A -85,B 0,C 180,E1 -14619.195,E2 -14619.195} C_VEL
LIN {X 0,Y 333.624,Z 156.925,A -85,B 0,C 180,E1 -14622.498,E2 -14622.498} C_VEL
LIN {X 0,Y 333.59,Z 156.928,A -85,B 0,C 180,E1 -14625.953,E2 -14625.953} C_VEL
LIN {X 0,Y 333.598,Z 156.931,A -85,B 0,C 180,E1 -14629.323,E2 -14629.323} C_VEL
LIN {X 0,Y 333.657,Z 156.923,A -85,B 0,C 180,E1 -14633.168,E2 -14633.168} C_VEL
LIN {X 0,Y 333.668,Z 156.92,A -85,B 0,C 180,E1 -14635.34,E2 -14635.34} C_VEL
LIN {X 0,Y 333.624,Z 156.925,A -85,B 0,C 180,E1 -14638.221,E2 -14638.221} C_VEL
LIN {X 0,Y 333.645,Z 156.924,A -85,B 0,C 180,E1 -14641.021,E2 -14641.021} C_VEL
LIN {X 0,Y 333.657,Z 156.922,A -85,B 0,C 180,E1 -14645.085,E2 -14645.085} C_VEL
LIN {X 0,Y 333.645,Z 156.924,A -85,B 0,C 180,E1 -14649.016,E2 -14649.016} C_VEL
LIN {X 0,Y 333.705,Z 156.914,A -85,B 0,C 180,E1 -14651.584,E2 -14651.584} C_VEL
LIN {X 0,Y 333.767,Z 156.906,A -85,B 0,C 180,E1 -14655.6,E2 -14655.6} C_VEL
LIN {X 0,Y 333.806,Z 156.902,A -85,B 0,C 180,E1 -14659.077,E2 -14659.077} C_VEL
LIN {X 0,Y 333.949,Z 156.886,A -85,B 0,C 180,E1 -14662.746,E2 -14662.746} C_VEL
LIN {X 0,Y 333.769,Z 156.907,A -85,B 0,C 180,E1 -14665.168,E2 -14665.168} C_VEL
LIN {X 0,Y 333.813,Z 157.096,A -85,B 0,C 180,E1 -14666.303,E2 -14666.303} C_VEL
LIN {X 0,Y 335.343,Z 163.661,A -85,B 0,C 180,E1 -14668.305,E2 -14668.305} C_VEL
LIN {X 0,Y 335.43,Z 164.118,A -85,B 0,C 180,E1 -14668.408,E2 -14668.408} C_VEL
LIN {X 0,Y 341.115,Z 180.611,A -85,B 0,C 180,E1 -14669.174,E2 -14669.174} C_VEL
LIN {X 0,Y 343.484,Z 192.437,A -85,B 0,C 180,E1 -14669.596,E2 -14669.596} C_VEL
LIN {X 0,Y 341.69,Z 271.297,A -85,B 0,C 180,E1 -14671.289,E2 -14671.289} C_VEL
LIN {X 0,Y 341.054,Z 284.595,A -85,B 0,C 180,E1 -14671.808,E2 -14671.808} C_VEL
LIN {X 0,Y 340.383,Z 296.699,A -85,B 0,C 180,E1 -14672.514,E2 -14672.514} C_VEL
LIN {X 0,Y 339.481,Z 308.213,A -85,B 0,C 180,E1 -14673.412,E2 -14673.412} C_VEL
LIN {X 0,Y 338.384,Z 319.154,A -85,B 0,C 180,E1 -14674.511,E2 -14674.511} C_VEL
LIN {X 0,Y 337.239,Z 329.626,A -85,B 0,C 180,E1 -14675.831,E2 -14675.831} C_VEL
LIN {X 0,Y 336.201,Z 338.483,A -85,B 0,C 180,E1 -14677.205,E2 -14677.205} C_VEL
LIN {X 0,Y 335.048,Z 347.391,A -85,B 0,C 180,E1 -14678.9,E2 -14678.9} C_VEL
LIN {X 0,Y 334.109,Z 354.587,A -85,B 0,C 180,E1 -14680.606,E2 -14680.606} C_VEL
LIN {X 0,Y 333.453,Z 359.987,A -85,B 0,C 180,E1 -14682.167,E2 -14682.167} C_VEL
LIN {X 0,Y 332.802,Z 365.465,A -85,B 0,C 180,E1 -14684.166,E2 -14684.166} C_VEL
LIN {X 0,Y 332.402,Z 369.216,A -85,B 0,C 180,E1 -14685.953,E2 -14685.953} C_VEL
LIN {X 0,Y 332.076,Z 372.005,A -85,B 0,C 180,E1 -14687.759,E2 -14687.759} C_VEL
LIN {X 0,Y 331.837,Z 374.025,A -85,B 0,C 180,E1 -14689.808,E2 -14689.808} C_VEL
LIN {X 0,Y 331.807,Z 374.778,A -85,B 0,C 180,E1 -14691.26,E2 -14691.26} C_VEL
LIN {X 0,Y 331.805,Z 374.968,A -85,B 0,C 180,E1 -14692.412,E2 -14692.412} C_VEL
LIN {X 0,Y 331.94,Z 374.415,A -85,B 0,C 180,E1 -14694.44,E2 -14694.44} C_VEL
LIN {X 0,Y 332.144,Z 372.851,A -85,B 0,C 180,E1 -14696.382,E2 -14696.382} C_VEL
LIN {X 0,Y 332.54,Z 370.106,A -85,B 0,C 180,E1 -14698.393,E2 -14698.393} C_VEL
LIN {X 0,Y 333.083,Z 366.101,A -85,B 0,C 180,E1 -14700.424,E2 -14700.424} C_VEL
LIN {X 0,Y 333.743,Z 361.375,A -85,B 0,C 180,E1 -14702.233,E2 -14702.233} C_VEL
LIN {X 0,Y 334.708,Z 354.915,A -85,B 0,C 180,E1 -14704.172,E2 -14704.172} C_VEL
LIN {X 0,Y 335.827,Z 347.811,A -85,B 0,C 180,E1 -14705.871,E2 -14705.871} C_VEL
LIN {X 0,Y 337.141,Z 338.71,A -85,B 0,C 180,E1 -14707.616,E2 -14707.616} C_VEL
LIN {X 0,Y 338.475,Z 329.061,A -85,B 0,C 180,E1 -14709.102,E2 -14709.102} C_VEL
LIN {X 0,Y 339.79,Z 318.712,A -85,B 0,C 180,E1 -14710.386,E2 -14710.386} C_VEL
LIN {X 0,Y 340.97,Z 308.012,A -85,B 0,C 180,E1 -14711.442,E2 -14711.442} C_VEL
LIN {X 0,Y 341.564,Z 301.962,A -85,B 0,C 180,E1 -14711.933,E2 -14711.933} C_VEL
LIN {X 0,Y 341.424,Z 296.622,A -85,B 0,C 180,E1 -14712.359,E2 -14712.359} C_VEL
LIN {X 0,Y 339.446,Z 287.889,A -85,B 0,C 180,E1 -14713.073,E2 -14713.073} C_VEL
LIN {X 0,Y 337.292,Z 278.943,A -85,B 0,C 180,E1 -14713.687,E2 -14713.687} C_VEL
LIN {X 0,Y 336.778,Z 273.274,A -85,B 0,C 180,E1 -14713.948,E2 -14713.948} C_VEL
LIN {X 0,Y 337.84,Z 234.082,A -85,B 0,C 180,E1 -14714.839,E2 -14714.839} C_VEL
LIN {X 0,Y 338.79,Z 193.303,A -85,B 0,C 180,E1 -14715.733,E2 -14715.733} C_VEL
LIN {X 0,Y 337.055,Z 185.808,A -85,B 0,C 180,E1 -14716.058,E2 -14716.058} C_VEL
LIN {X 0,Y 329.66,Z 167.975,A -85,B 0,C 180,E1 -14717.142,E2 -14717.142} C_VEL
LIN {X 0,Y 328.287,Z 164.802,A -85,B 0,C 180,E1 -14717.39,E2 -14717.39} C_VEL
LIN {X 0,Y 326.648,Z 157.804,A -85,B 0,C 180,E1 -14719.728,E2 -14719.728} C_VEL
LIN {X 0,Y 326.629,Z 157.804,A -85,B 0,C 180,E1 -14722.954,E2 -14722.954} C_VEL
LIN {X 0,Y 326.604,Z 157.803,A -85,B 0,C 180,E1 -14725.982,E2 -14725.982} C_VEL
LIN {X 0,Y 326.658,Z 157.791,A -85,B 0,C 180,E1 -14730.342,E2 -14730.342} C_VEL
LIN {X 0,Y 326.688,Z 157.794,A -85,B 0,C 180,E1 -14734.517,E2 -14734.517} C_VEL
LIN {X 0,Y 326.644,Z 157.796,A -85,B 0,C 180,E1 -14738.546,E2 -14738.546} C_VEL
LIN {X 0,Y 326.706,Z 157.791,A -85,B 0,C 180,E1 -14741.176,E2 -14741.176} C_VEL
LIN {X 0,Y 326.763,Z 157.779,A -85,B 0,C 180,E1 -14745.434,E2 -14745.434} C_VEL
LIN {X 0,Y 326.759,Z 157.785,A -85,B 0,C 180,E1 -14748.84,E2 -14748.84} C_VEL
LIN {X 0,Y 326.919,Z 157.759,A -85,B 0,C 180,E1 -14752.59,E2 -14752.59} C_VEL
LIN {X 0,Y 326.764,Z 157.771,A -85,B 0,C 180,E1 -14755.066,E2 -14755.066} C_VEL
LIN {X 0,Y 327.043,Z 157.741,A -85,B 0,C 180,E1 -14757.538,E2 -14757.538} C_VEL
LIN {X 0,Y 327.141,Z 157.724,A -85,B 0,C 180,E1 -14760.001,E2 -14760.001} C_VEL
LIN {X 0,Y 327.012,Z 157.745,A -85,B 0,C 180,E1 -14762.465,E2 -14762.465} C_VEL
LIN {X 0,Y 326.946,Z 157.745,A -85,B 0,C 180,E1 -14766.171,E2 -14766.171} C_VEL
LIN {X 0,Y 326.785,Z 157.771,A -85,B 0,C 180,E1 -14769.908,E2 -14769.908} C_VEL
LIN {X 0,Y 326.758,Z 157.783,A -85,B 0,C 180,E1 -14773.686,E2 -14773.686} C_VEL
LIN {X 0,Y 326.644,Z 157.789,A -85,B 0,C 180,E1 -14777.532,E2 -14777.532} C_VEL
LIN {X 0,Y 326.613,Z 157.796,A -85,B 0,C 180,E1 -14780.139,E2 -14780.139} C_VEL
LIN {X 0,Y 326.593,Z 157.799,A -85,B 0,C 180,E1 -14782.79,E2 -14782.79} C_VEL
LIN {X 0,Y 326.599,Z 157.794,A -85,B 0,C 180,E1 -14786.866,E2 -14786.866} C_VEL
LIN {X 0,Y 326.613,Z 157.791,A -85,B 0,C 180,E1 -14790.603,E2 -14790.603} C_VEL
LIN {X 0,Y 326.608,Z 157.795,A -85,B 0,C 180,E1 -14794.02,E2 -14794.02} C_VEL
LIN {X 0,Y 326.624,Z 157.797,A -85,B 0,C 180,E1 -14797.238,E2 -14797.238} C_VEL
LIN {X 0,Y 326.545,Z 157.808,A -85,B 0,C 180,E1 -14801.125,E2 -14801.125} C_VEL
LIN {X 0,Y 326.561,Z 157.808,A -85,B 0,C 180,E1 -14803.527,E2 -14803.527} C_VEL
LIN {X 0,Y 326.574,Z 157.809,A -85,B 0,C 180,E1 -14807.03,E2 -14807.03} C_VEL
LIN {X 0,Y 326.574,Z 157.807,A -85,B 0,C 180,E1 -14810.782,E2 -14810.782} C_VEL
LIN {X 0,Y 326.615,Z 157.8,A -85,B 0,C 180,E1 -14814.481,E2 -14814.481} C_VEL
LIN {X 0,Y 326.607,Z 157.906,A -85,B 0,C 180,E1 -14817.105,E2 -14817.105} C_VEL
LIN {X 0,Y 329.1,Z 168.232,A -85,B 0,C 180,E1 -14820.231,E2 -14820.231} C_VEL
LIN {X 0,Y 331.431,Z 179.929,A -85,B 0,C 180,E1 -14823.557,E2 -14823.557} C_VEL
LIN {X 0,Y 331.334,Z 183.832,A -85,B 0,C 180,E1 -14824.563,E2 -14824.563} C_VEL
LIN {X 0,Y 331.129,Z 185.485,A -85,B 0,C 180,E1 -14824.949,E2 -14824.949} C_VEL
LIN {X 0,Y 335.736,Z 209.714,A -85,B 0,C 180,E1 -14825.934,E2 -14825.934} C_VEL
LIN {X 0,Y 338.144,Z 226.9,A -85,B 0,C 180,E1 -14826.541,E2 -14826.541} C_VEL
LIN {X 0,Y 336.54,Z 294.321,A -85,B 0,C 180,E1 -14828.041,E2 -14828.041} C_VEL
LIN {X 0,Y 335.616,Z 308.148,A -85,B 0,C 180,E1 -14828.583,E2 -14828.583} C_VEL
LIN {X 0,Y 334.47,Z 320.608,A -85,B 0,C 180,E1 -14829.313,E2 -14829.313} C_VEL
LIN {X 0,Y 333.193,Z 332.539,A -85,B 0,C 180,E1 -14830.276,E2 -14830.276} C_VEL
LIN {X 0,Y 331.679,Z 343.998,A -85,B 0,C 180,E1 -14831.468,E2 -14831.468} C_VEL
LIN {X 0,Y 330.169,Z 354.353,A -85,B 0,C 180,E1 -14832.822,E2 -14832.822} C_VEL
LIN {X 0,Y 328.999,Z 363.444,A -85,B 0,C 180,E1 -14834.31,E2 -14834.31} C_VEL
LIN {X 0,Y 327.742,Z 372.042,A -85,B 0,C 180,E1 -14836.04,E2 -14836.04} C_VEL
LIN {X 0,Y 326.508,Z 379.47,A -85,B 0,C 180,E1 -14837.886,E2 -14837.886} C_VEL
LIN {X 0,Y 325.704,Z 386.325,A -85,B 0,C 180,E1 -14840.06,E2 -14840.06} C_VEL
LIN {X 0,Y 325.213,Z 390.86,A -85,B 0,C 180,E1 -14841.925,E2 -14841.925} C_VEL
LIN {X 0,Y 324.904,Z 395.048,A -85,B 0,C 180,E1 -14844.289,E2 -14844.289} C_VEL
LIN {X 0,Y 324.9,Z 397.368,A -85,B 0,C 180,E1 -14846.279,E2 -14846.279} C_VEL
LIN {X 0,Y 324.86,Z 398.294,A -85,B 0,C 180,E1 -14847.52,E2 -14847.52} C_VEL
LIN {X 0,Y 324.88,Z 398.796,A -85,B 0,C 180,E1 -14848.761,E2 -14848.761} C_VEL
LIN {X 0,Y 324.95,Z 398.883,A -85,B 0,C 180,E1 -14850,E2 -14850} C_VEL
LIN {X 0,Y 324.894,Z 398.575,A -85,B 0,C 180,E1 -14851.24,E2 -14851.24} C_VEL
LIN {X 0,Y 324.862,Z 397.877,A -85,B 0,C 180,E1 -14852.48,E2 -14852.48} C_VEL
LIN {X 0,Y 324.9,Z 396.754,A -85,B 0,C 180,E1 -14853.721,E2 -14853.721} C_VEL
LIN {X 0,Y 324.906,Z 394.051,A -85,B 0,C 180,E1 -14855.714,E2 -14855.714} C_VEL
LIN {X 0,Y 325.113,Z 390.764,A -85,B 0,C 180,E1 -14857.453,E2 -14857.453} C_VEL
LIN {X 0,Y 325.493,Z 386.147,A -85,B 0,C 180,E1 -14859.32,E2 -14859.32} C_VEL
LIN {X 0,Y 326.162,Z 379.141,A -85,B 0,C 180,E1 -14861.497,E2 -14861.497} C_VEL
LIN {X 0,Y 327.183,Z 371.564,A -85,B 0,C 180,E1 -14863.351,E2 -14863.351} C_VEL
LIN {X 0,Y 328.167,Z 363.817,A -85,B 0,C 180,E1 -14864.892,E2 -14864.892} C_VEL
LIN {X 0,Y 329.265,Z 354.361,A -85,B 0,C 180,E1 -14866.429,E2 -14866.429} C_VEL
LIN {X 0,Y 330.495,Z 343.86,A -85,B 0,C 180,E1 -14867.8,E2 -14867.8} C_VEL
LIN {X 0,Y 331.821,Z 332.201,A -85,B 0,C 180,E1 -14869.005,E2 -14869.005} C_VEL
LIN {X 0,Y 333.049,Z 319.82,A -85,B 0,C 180,E1 -14869.974,E2 -14869.974} C_VEL
LIN {X 0,Y 334.1,Z 306.817,A -85,B 0,C 180,E1 -14870.712,E2 -14870.712} C_VEL
LIN {X 0,Y 334.783,Z 294.176,A -85,B 0,C 180,E1 -14871.191,E2 -14871.191} C_VEL
LIN {X 0,Y 336.177,Z 225.226,A -85,B 0,C 180,E1 -14872.71,E2 -14872.71} C_VEL
LIN {X 0,Y 330.618,Z 189.162,A -85,B 0,C 180,E1 -14873.926,E2 -14873.926} C_VEL
LIN {X 0,Y 330.216,Z 186.233,A -85,B 0,C 180,E1 -14874.047,E2 -14874.047} C_VEL
LIN {X 0,Y 330.888,Z 179.149,A -85,B 0,C 180,E1 -14875.812,E2 -14875.812} C_VEL
LIN {X 0,Y 329.06,Z 168.892,A -85,B 0,C 180,E1 -14878.612,E2 -14878.612} C_VEL
LIN {X 0,Y 326.623,Z 157.801,A -85,B 0,C 180,E1 -14881.815,E2 -14881.815} C_VEL
LIN {X 0,Y 326.617,Z 157.802,A -85,B 0,C 180,E1 -14885.52,E2 -14885.52} C_VEL
LIN {X 0,Y 326.591,Z 157.803,A -85,B 0,C 180,E1 -14889.221,E2 -14889.221} C_VEL
LIN {X 0,Y 326.577,Z 157.803,A -85,B 0,C 180,E1 -14892.971,E2 -14892.971} C_VEL
LIN {X 0,Y 326.578,Z 157.806,A -85,B 0,C 180,E1 -14897.029,E2 -14897.029} C_VEL
LIN {X 0,Y 326.587,Z 157.805,A -85,B 0,C 180,E1 -14901.385,E2 -14901.385} C_VEL
LIN {X 0,Y 326.623,Z 157.8,A -85,B 0,C 180,E1 -14904.851,E2 -14904.851} C_VEL
LIN {X 0,Y 326.613,Z 157.8,A -85,B 0,C 180,E1 -14907.455,E2 -14907.455} C_VEL
LIN {X 0,Y 326.621,Z 157.798,A -85,B 0,C 180,E1 -14910.336,E2 -14910.336} C_VEL
LIN {X 0,Y 326.647,Z 157.797,A -85,B 0,C 180,E1 -14914.644,E2 -14914.644} C_VEL
LIN {X 0,Y 326.615,Z 157.801,A -85,B 0,C 180,E1 -14918.542,E2 -14918.542} C_VEL
LIN {X 0,Y 326.653,Z 157.794,A -85,B 0,C 180,E1 -14921.205,E2 -14921.205} C_VEL
LIN {X 0,Y 326.73,Z 157.783,A -85,B 0,C 180,E1 -14925.458,E2 -14925.458} C_VEL
LIN {X 0,Y 326.762,Z 157.781,A -85,B 0,C 180,E1 -14928.838,E2 -14928.838} C_VEL
LIN {X 0,Y 326.918,Z 157.761,A -85,B 0,C 180,E1 -14932.588,E2 -14932.588} C_VEL
LIN {X 0,Y 326.751,Z 157.78,A -85,B 0,C 180,E1 -14935.063,E2 -14935.063} C_VEL
LIN {X 0,Y 327.013,Z 157.748,A -85,B 0,C 180,E1 -14937.535,E2 -14937.535} C_VEL
LIN {X 0,Y 327.033,Z 157.744,A -85,B 0,C 180,E1 -14941.23,E2 -14941.23} C_VEL
LIN {X 0,Y 326.752,Z 157.778,A -85,B 0,C 180,E1 -14943.699,E2 -14943.699} C_VEL
LIN {X 0,Y 326.923,Z 157.76,A -85,B 0,C 180,E1 -14946.463,E2 -14946.463} C_VEL
LIN {X 0,Y 326.784,Z 157.781,A -85,B 0,C 180,E1 -14949.906,E2 -14949.906} C_VEL
LIN {X 0,Y 326.744,Z 157.784,A -85,B 0,C 180,E1 -14953.685,E2 -14953.685} C_VEL
LIN {X 0,Y 326.628,Z 157.796,A -85,B 0,C 180,E1 -14957.531,E2 -14957.531} C_VEL
LIN {X 0,Y 326.607,Z 157.802,A -85,B 0,C 180,E1 -14961.456,E2 -14961.456} C_VEL
LIN {X 0,Y 326.599,Z 157.803,A -85,B 0,C 180,E1 -14965.49,E2 -14965.49} C_VEL
LIN {X 0,Y 326.59,Z 157.798,A -85,B 0,C 180,E1 -14968.256,E2 -14968.256} C_VEL
LIN {X 0,Y 326.572,Z 157.804,A -85,B 0,C 180,E1 -14971.096,E2 -14971.096} C_VEL
LIN {X 0,Y 326.606,Z 157.799,A -85,B 0,C 180,E1 -14974.018,E2 -14974.018} C_VEL
LIN {X 0,Y 326.621,Z 157.8,A -85,B 0,C 180,E1 -14977.236,E2 -14977.236} C_VEL
LIN {X 0,Y 326.541,Z 157.81,A -85,B 0,C 180,E1 -14981.123,E2 -14981.123} C_VEL
LIN {X 0,Y 326.556,Z 157.807,A -85,B 0,C 180,E1 -14983.525,E2 -14983.525} C_VEL
LIN {X 0,Y 326.569,Z 157.806,A -85,B 0,C 180,E1 -14987.028,E2 -14987.028} C_VEL
LIN {X 0,Y 326.577,Z 157.805,A -85,B 0,C 180,E1 -14991.384,E2 -14991.384} C_VEL
LIN {X 0,Y 326.613,Z 157.802,A -85,B 0,C 180,E1 -14994.851,E2 -14994.851} C_VEL
LIN {X 0,Y 326.603,Z 157.8,A -85,B 0,C 180,E1 -14997.454,E2 -14997.454} C_VEL
LIN {X 0,Y 326.609,Z 157.8,A -85,B 0,C 180,E1 -15000.335,E2 -15000.335} C_VEL
LIN {X 0,Y 326.594,Z 157.804,A -85,B 0,C 180,E1 -15004.508,E2 -15004.508} C_VEL
LIN {X 0,Y 326.602,Z 157.804,A -85,B 0,C 180,E1 -15008.542,E2 -15008.542} C_VEL
LIN {X 0,Y 326.641,Z 157.795,A -85,B 0,C 180,E1 -15011.205,E2 -15011.205} C_VEL
LIN {X 0,Y 326.718,Z 157.784,A -85,B 0,C 180,E1 -15015.459,E2 -15015.459} C_VEL
LIN {X 0,Y 326.747,Z 157.782,A -85,B 0,C 180,E1 -15018.838,E2 -15018.838} C_VEL
LIN {X 0,Y 326.906,Z 157.764,A -85,B 0,C 180,E1 -15022.588,E2 -15022.588} C_VEL
LIN {X 0,Y 326.739,Z 157.783,A -85,B 0,C 180,E1 -15025.064,E2 -15025.064} C_VEL
LIN {X 0,Y 326.744,Z 157.892,A -85,B 0,C 180,E1 -15025.914,E2 -15025.914} C_VEL
LIN {X 0,Y 328.298,Z 164.393,A -85,B 0,C 180,E1 -15027.909,E2 -15027.909} C_VEL
LIN {X 0,Y 334.624,Z 182.262,A -85,B 0,C 180,E1 -15028.778,E2 -15028.778} C_VEL
LIN {X 0,Y 336.833,Z 193.849,A -85,B 0,C 180,E1 -15029.196,E2 -15029.196} C_VEL
LIN {X 0,Y 334.978,Z 271.712,A -85,B 0,C 180,E1 -15030.901,E2 -15030.901} C_VEL
LIN {X 0,Y 334.339,Z 284.932,A -85,B 0,C 180,E1 -15031.43,E2 -15031.43} C_VEL
LIN {X 0,Y 333.582,Z 297.6,A -85,B 0,C 180,E1 -15032.188,E2 -15032.188} C_VEL
LIN {X 0,Y 332.583,Z 309.723,A -85,B 0,C 180,E1 -15033.18,E2 -15033.18} C_VEL
LIN {X 0,Y 331.406,Z 321.273,A -85,B 0,C 180,E1 -15034.401,E2 -15034.401} C_VEL
LIN {X 0,Y 330.166,Z 331.8,A -85,B 0,C 180,E1 -15035.803,E2 -15035.803} C_VEL
LIN {X 0,Y 328.973,Z 341.166,A -85,B 0,C 180,E1 -15037.364,E2 -15037.364} C_VEL
LIN {X 0,Y 327.876,Z 349.189,A -85,B 0,C 180,E1 -15039.006,E2 -15039.006} C_VEL
LIN {X 0,Y 326.922,Z 356.453,A -85,B 0,C 180,E1 -15040.842,E2 -15040.842} C_VEL
LIN {X 0,Y 326.275,Z 361.556,A -85,B 0,C 180,E1 -15042.439,E2 -15042.439} C_VEL
LIN {X 0,Y 325.668,Z 366.509,A -85,B 0,C 180,E1 -15044.374,E2 -15044.374} C_VEL
LIN {X 0,Y 325.217,Z 370.266,A -85,B 0,C 180,E1 -15046.316,E2 -15046.316} C_VEL
LIN {X 0,Y 324.958,Z 372.5,A -85,B 0,C 180,E1 -15047.902,E2 -15047.902} C_VEL
LIN {X 0,Y 324.735,Z 374.589,A -85,B 0,C 180,E1 -15050.26,E2 -15050.26} C_VEL
LIN {X 0,Y 324.712,Z 375.116,A -85,B 0,C 180,E1 -15051.589,E2 -15051.589} C_VEL
LIN {X 0,Y 324.745,Z 375.176,A -85,B 0,C 180,E1 -15052.926,E2 -15052.926} C_VEL
LIN {X 0,Y 324.873,Z 374.574,A -85,B 0,C 180,E1 -15054.692,E2 -15054.692} C_VEL
LIN {X 0,Y 325.191,Z 372.563,A -85,B 0,C 180,E1 -15056.991,E2 -15056.991} C_VEL
LIN {X 0,Y 325.611,Z 369.549,A -85,B 0,C 180,E1 -15059.054,E2 -15059.054} C_VEL
LIN {X 0,Y 326.239,Z 365.253,A -85,B 0,C 180,E1 -15061.132,E2 -15061.132} C_VEL
LIN {X 0,Y 327.264,Z 358.744,A -85,B 0,C 180,E1 -15063.435,E2 -15063.435} C_VEL
LIN {X 0,Y 328.324,Z 351.933,A -85,B 0,C 180,E1 -15065.307,E2 -15065.307} C_VEL
LIN {X 0,Y 329.563,Z 344.051,A -85,B 0,C 180,E1 -15067.045,E2 -15067.045} C_VEL
LIN {X 0,Y 331.045,Z 334.18,A -85,B 0,C 180,E1 -15068.775,E2 -15068.775} C_VEL
LIN {X 0,Y 332.568,Z 323.614,A -85,B 0,C 180,E1 -15070.252,E2 -15070.252} C_VEL
LIN {X 0,Y 333.914,Z 312.028,A -85,B 0,C 180,E1 -15071.528,E2 -15071.528} C_VEL
LIN {X 0,Y 335.138,Z 300.278,A -85,B 0,C 180,E1 -15072.529,E2 -15072.529} C_VEL
LIN {X 0,Y 336.038,Z 288.125,A -85,B 0,C 180,E1 -15073.313,E2 -15073.313} C_VEL
LIN {X 0,Y 336.716,Z 274.848,A -85,B 0,C 180,E1 -15073.896,E2 -15073.896} C_VEL
LIN {X 0,Y 336.778,Z 273.274,A -85,B 0,C 180,E1 -15073.948,E2 -15073.948} C_VEL
LIN {X 0,Y 336.275,Z 267.531,A -85,B 0,C 180,E1 -15074.177,E2 -15074.177} C_VEL
LIN {X 0,Y 331.639,Z 248.859,A -85,B 0,C 180,E1 -15074.991,E2 -15074.991} C_VEL
LIN {X 0,Y 331.196,Z 243.056,A -85,B 0,C 180,E1 -15075.16,E2 -15075.16} C_VEL
LIN {X 0,Y 332.368,Z 194.121,A -85,B 0,C 180,E1 -15076.255,E2 -15076.255} C_VEL
LIN {X 0,Y 330.926,Z 188.242,A -85,B 0,C 180,E1 -15076.525,E2 -15076.525} C_VEL
LIN {X 0,Y 323.796,Z 171.103,A -85,B 0,C 180,E1 -15077.609,E2 -15077.609} C_VEL
LIN {X 0,Y 321.174,Z 165.201,A -85,B 0,C 180,E1 -15078.029,E2 -15078.029} C_VEL
LIN {X 0,Y 319.599,Z 158.677,A -85,B 0,C 180,E1 -15080.258,E2 -15080.258} C_VEL
LIN {X 0,Y 319.556,Z 158.687,A -85,B 0,C 180,E1 -15083.574,E2 -15083.574} C_VEL
LIN {X 0,Y 319.574,Z 158.677,A -85,B 0,C 180,E1 -15086.688,E2 -15086.688} C_VEL
LIN {X 0,Y 319.588,Z 158.676,A -85,B 0,C 180,E1 -15089.618,E2 -15089.618} C_VEL
LIN {X 0,Y 319.607,Z 158.673,A -85,B 0,C 180,E1 -15092.499,E2 -15092.499} C_VEL
LIN {X 0,Y 319.603,Z 158.673,A -85,B 0,C 180,E1 -15095.305,E2 -15095.305} C_VEL
LIN {X 0,Y 319.595,Z 158.675,A -85,B 0,C 180,E1 -15098.049,E2 -15098.049} C_VEL
LIN {X 0,Y 319.656,Z 158.671,A -85,B 0,C 180,E1 -15100.98,E2 -15100.98} C_VEL
LIN {X 0,Y 319.711,Z 158.659,A -85,B 0,C 180,E1 -15105.29,E2 -15105.29} C_VEL
LIN {X 0,Y 319.715,Z 158.66,A -85,B 0,C 180,E1 -15108.591,E2 -15108.591} C_VEL
LIN {X 0,Y 319.857,Z 158.636,A -85,B 0,C 180,E1 -15112.426,E2 -15112.426} C_VEL
LIN {X 0,Y 319.732,Z 158.647,A -85,B 0,C 180,E1 -15114.957,E2 -15114.957} C_VEL
LIN {X 0,Y 319.986,Z 158.62,A -85,B 0,C 180,E1 -15117.483,E2 -15117.483} C_VEL
LIN {X 0,Y 320.096,Z 158.602,A -85,B 0,C 180,E1 -15120.001,E2 -15120.001} C_VEL
LIN {X 0,Y 319.959,Z 158.624,A -85,B 0,C 180,E1 -15122.519,E2 -15122.519} C_VEL
LIN {X 0,Y 319.903,Z 158.623,A -85,B 0,C 180,E1 -15126.307,E2 -15126.307} C_VEL
LIN {X 0,Y 319.737,Z 158.646,A -85,B 0,C 180,E1 -15130.129,E2 -15130.129} C_VEL
LIN {X 0,Y 319.731,Z 158.659,A -85,B 0,C 180,E1 -15133.993,E2 -15133.993} C_VEL
LIN {X 0,Y 319.602,Z 158.671,A -85,B 0,C 180,E1 -15137.931,E2 -15137.931} C_VEL
LIN {X 0,Y 319.565,Z 158.67,A -85,B 0,C 180,E1 -15141.956,E2 -15141.956} C_VEL
LIN {X 0,Y 319.552,Z 158.67,A -85,B 0,C 180,E1 -15146.096,E2 -15146.096} C_VEL
LIN {X 0,Y 319.543,Z 158.682,A -85,B 0,C 180,E1 -15148.939,E2 -15148.939} C_VEL
LIN {X 0,Y 319.526,Z 158.684,A -85,B 0,C 180,E1 -15151.863,E2 -15151.863} C_VEL
LIN {X 0,Y 319.58,Z 158.675,A -85,B 0,C 180,E1 -15155.543,E2 -15155.543} C_VEL
LIN {X 0,Y 319.531,Z 158.685,A -85,B 0,C 180,E1 -15159.663,E2 -15159.663} C_VEL
LIN {X 0,Y 319.521,Z 158.686,A -85,B 0,C 180,E1 -15163.46,E2 -15163.46} C_VEL
LIN {X 0,Y 319.553,Z 158.684,A -85,B 0,C 180,E1 -15167.016,E2 -15167.016} C_VEL
LIN {X 0,Y 319.517,Z 158.688,A -85,B 0,C 180,E1 -15170.367,E2 -15170.367} C_VEL
LIN {X 0,Y 319.582,Z 158.675,A -85,B 0,C 180,E1 -15174.458,E2 -15174.458} C_VEL
LIN {X 0,Y 319.598,Z 158.817,A -85,B 0,C 180,E1 -15176.556,E2 -15176.556} C_VEL
LIN {X 0,Y 322.152,Z 169.486,A -85,B 0,C 180,E1 -15179.883,E2 -15179.883} C_VEL
LIN {X 0,Y 324.259,Z 179.872,A -85,B 0,C 180,E1 -15182.925,E2 -15182.925} C_VEL
LIN {X 0,Y 324.641,Z 183.767,A -85,B 0,C 180,E1 -15183.999,E2 -15183.999} C_VEL
LIN {X 0,Y 324.478,Z 185.063,A -85,B 0,C 180,E1 -15184.33,E2 -15184.33} C_VEL
LIN {X 0,Y 329.394,Z 210.933,A -85,B 0,C 180,E1 -15185.427,E2 -15185.427} C_VEL
LIN {X 0,Y 331.693,Z 226.629,A -85,B 0,C 180,E1 -15186.006,E2 -15186.006} C_VEL
LIN {X 0,Y 330.052,Z 294.225,A -85,B 0,C 180,E1 -15187.545,E2 -15187.545} C_VEL
LIN {X 0,Y 329.1,Z 307.988,A -85,B 0,C 180,E1 -15188.096,E2 -15188.096} C_VEL
LIN {X 0,Y 327.856,Z 320.924,A -85,B 0,C 180,E1 -15188.876,E2 -15188.876} C_VEL
LIN {X 0,Y 326.536,Z 332.697,A -85,B 0,C 180,E1 -15189.857,E2 -15189.857} C_VEL
LIN {X 0,Y 324.961,Z 344.066,A -85,B 0,C 180,E1 -15191.07,E2 -15191.07} C_VEL
LIN {X 0,Y 323.377,Z 354.448,A -85,B 0,C 180,E1 -15192.466,E2 -15192.466} C_VEL
LIN {X 0,Y 322.079,Z 363.826,A -85,B 0,C 180,E1 -15194.054,E2 -15194.054} C_VEL
LIN {X 0,Y 320.844,Z 371.94,A -85,B 0,C 180,E1 -15195.734,E2 -15195.734} C_VEL
LIN {X 0,Y 319.542,Z 379.34,A -85,B 0,C 180,E1 -15197.617,E2 -15197.617} C_VEL
LIN {X 0,Y 318.663,Z 386.158,A -85,B 0,C 180,E1 -15199.838,E2 -15199.838} C_VEL
LIN {X 0,Y 318.171,Z 390.673,A -85,B 0,C 180,E1 -15201.745,E2 -15201.745} C_VEL
LIN {X 0,Y 317.89,Z 394.11,A -85,B 0,C 180,E1 -15203.654,E2 -15203.654} C_VEL
LIN {X 0,Y 317.807,Z 397.142,A -85,B 0,C 180,E1 -15206.196,E2 -15206.196} C_VEL
LIN {X 0,Y 317.78,Z 398.058,A -85,B 0,C 180,E1 -15207.465,E2 -15207.465} C_VEL
LIN {X 0,Y 317.789,Z 398.541,A -85,B 0,C 180,E1 -15208.733,E2 -15208.733} C_VEL
LIN {X 0,Y 317.854,Z 398.618,A -85,B 0,C 180,E1 -15210,E2 -15210} C_VEL
LIN {X 0,Y 317.802,Z 398.3,A -85,B 0,C 180,E1 -15211.267,E2 -15211.267} C_VEL
LIN {X 0,Y 317.781,Z 397.593,A -85,B 0,C 180,E1 -15212.535,E2 -15212.535} C_VEL
LIN {X 0,Y 317.807,Z 396.448,A -85,B 0,C 180,E1 -15213.804,E2 -15213.804} C_VEL
LIN {X 0,Y 317.805,Z 394.051,A -85,B 0,C 180,E1 -15215.644,E2 -15215.644} C_VEL
LIN {X 0,Y 318.035,Z 390.415,A -85,B 0,C 180,E1 -15217.62,E2 -15217.62} C_VEL
LIN {X 0,Y 318.436,Z 385.769,A -85,B 0,C 180,E1 -15219.528,E2 -15219.528} C_VEL
LIN {X 0,Y 319.178,Z 378.734,A -85,B 0,C 180,E1 -15221.752,E2 -15221.752} C_VEL
LIN {X 0,Y 320.242,Z 371.124,A -85,B 0,C 180,E1 -15223.646,E2 -15223.646} C_VEL
LIN {X 0,Y 321.267,Z 363.336,A -85,B 0,C 180,E1 -15225.219,E2 -15225.219} C_VEL
LIN {X 0,Y 322.408,Z 353.813,A -85,B 0,C 180,E1 -15226.788,E2 -15226.788} C_VEL
LIN {X 0,Y 323.694,Z 343.252,A -85,B 0,C 180,E1 -15228.187,E2 -15228.187} C_VEL
LIN {X 0,Y 325.114,Z 331.508,A -85,B 0,C 180,E1 -15229.413,E2 -15229.413} C_VEL
LIN {X 0,Y 326.357,Z 318.953,A -85,B 0,C 180,E1 -15230.402,E2 -15230.402} C_VEL
LIN {X 0,Y 327.45,Z 305.743,A -85,B 0,C 180,E1 -15231.152,E2 -15231.152} C_VEL
LIN {X 0,Y 328.139,Z 292.78,A -85,B 0,C 180,E1 -15231.63,E2 -15231.63} C_VEL
LIN {X 0,Y 329.456,Z 225.474,A -85,B 0,C 180,E1 -15233.144,E2 -15233.144} C_VEL
LIN {X 0,Y 323.704,Z 187.94,A -85,B 0,C 180,E1 -15234.445,E2 -15234.445} C_VEL
LIN {X 0,Y 323.41,Z 186.028,A -85,B 0,C 180,E1 -15234.525,E2 -15234.525} C_VEL
LIN {X 0,Y 323.894,Z 180.034,A -85,B 0,C 180,E1 -15236.06,E2 -15236.06} C_VEL
LIN {X 0,Y 322.193,Z 170.654,A -85,B 0,C 180,E1 -15238.678,E2 -15238.678} C_VEL
LIN {X 0,Y 319.573,Z 158.681,A -85,B 0,C 180,E1 -15242.229,E2 -15242.229} C_VEL
LIN {X 0,Y 319.561,Z 158.677,A -85,B 0,C 180,E1 -15246.428,E2 -15246.428} C_VEL
LIN {X 0,Y 319.533,Z 158.684,A -85,B 0,C 180,E1 -15249.662,E2 -15249.662} C_VEL
LIN {X 0,Y 319.523,Z 158.686,A -85,B 0,C 180,E1 -15253.46,E2 -15253.46} C_VEL
LIN {X 0,Y 319.556,Z 158.68,A -85,B 0,C 180,E1 -15257.016,E2 -15257.016} C_VEL
LIN {X 0,Y 319.55,Z 158.678,A -85,B 0,C 180,E1 -15260.37,E2 -15260.37} C_VEL
LIN {X 0,Y 319.583,Z 158.675,A -85,B 0,C 180,E1 -15264.457,E2 -15264.457} C_VEL
LIN {X 0,Y 319.529,Z 158.681,A -85,B 0,C 180,E1 -15268.137,E2 -15268.137} C_VEL
LIN {X 0,Y 319.576,Z 158.675,A -85,B 0,C 180,E1 -15271.603,E2 -15271.603} C_VEL
LIN {X 0,Y 319.577,Z 158.676,A -85,B 0,C 180,E1 -15275.301,E2 -15275.301} C_VEL
LIN {X 0,Y 319.568,Z 158.676,A -85,B 0,C 180,E1 -15278.045,E2 -15278.045} C_VEL
LIN {X 0,Y 319.592,Z 158.673,A -85,B 0,C 180,E1 -15282.068,E2 -15282.068} C_VEL
LIN {X 0,Y 319.714,Z 158.658,A -85,B 0,C 180,E1 -15286.006,E2 -15286.006} C_VEL
LIN {X 0,Y 319.74,Z 158.653,A -85,B 0,C 180,E1 -15289.871,E2 -15289.871} C_VEL
LIN {X 0,Y 319.904,Z 158.631,A -85,B 0,C 180,E1 -15293.693,E2 -15293.693} C_VEL
LIN {X 0,Y 319.959,Z 158.627,A -85,B 0,C 180,E1 -15297.481,E2 -15297.481} C_VEL
LIN {X 0,Y 320.002,Z 158.619,A -85,B 0,C 180,E1 -15301.257,E2 -15301.257} C_VEL
LIN {X 0,Y 319.702,Z 158.656,A -85,B 0,C 180,E1 -15303.78,E2 -15303.78} C_VEL
LIN {X 0,Y 319.888,Z 158.637,A -85,B 0,C 180,E1 -15306.445,E2 -15306.445} C_VEL
LIN {X 0,Y 319.736,Z 158.658,A -85,B 0,C 180,E1 -15310.127,E2 -15310.127} C_VEL
LIN {X 0,Y 319.711,Z 158.658,A -85,B 0,C 180,E1 -15313.992,E2 -15313.992} C_VEL
LIN {X 0,Y 319.584,Z 158.676,A -85,B 0,C 180,E1 -15317.93,E2 -15317.93} C_VEL
LIN {X 0,Y 319.562,Z 158.679,A -85,B 0,C 180,E1 -15321.953,E2 -15321.953} C_VEL
LIN {X 0,Y 319.549,Z 158.675,A -85,B 0,C 180,E1 -15326.094,E2 -15326.094} C_VEL
LIN {X 0,Y 319.524,Z 158.678,A -85,B 0,C 180,E1 -15328.939,E2 -15328.939} C_VEL
LIN {X 0,Y 319.523,Z 158.683,A -85,B 0,C 180,E1 -15331.861,E2 -15331.861} C_VEL
LIN {X 0,Y 319.578,Z 158.676,A -85,B 0,C 180,E1 -15335.541,E2 -15335.541} C_VEL
LIN {X 0,Y 319.525,Z 158.682,A -85,B 0,C 180,E1 -15339.661,E2 -15339.661} C_VEL
LIN {X 0,Y 319.515,Z 158.685,A -85,B 0,C 180,E1 -15343.459,E2 -15343.459} C_VEL
LIN {X 0,Y 319.547,Z 158.68,A -85,B 0,C 180,E1 -15347.015,E2 -15347.015} C_VEL
LIN {X 0,Y 319.541,Z 158.68,A -85,B 0,C 180,E1 -15350.369,E2 -15350.369} C_VEL
LIN {X 0,Y 319.573,Z 158.676,A -85,B 0,C 180,E1 -15354.456,E2 -15354.456} C_VEL
LIN {X 0,Y 319.519,Z 158.683,A -85,B 0,C 180,E1 -15358.136,E2 -15358.136} C_VEL
LIN {X 0,Y 319.563,Z 158.675,A -85,B 0,C 180,E1 -15361.603,E2 -15361.603} C_VEL
LIN {X 0,Y 319.52,Z 158.681,A -85,B 0,C 180,E1 -15365.297,E2 -15365.297} C_VEL
LIN {X 0,Y 319.556,Z 158.677,A -85,B 0,C 180,E1 -15368.044,E2 -15368.044} C_VEL
LIN {X 0,Y 319.58,Z 158.676,A -85,B 0,C 180,E1 -15372.068,E2 -15372.068} C_VEL
LIN {X 0,Y 319.702,Z 158.66,A -85,B 0,C 180,E1 -15376.006,E2 -15376.006} C_VEL
LIN {X 0,Y 319.726,Z 158.657,A -85,B 0,C 180,E1 -15379.872,E2 -15379.872} C_VEL
LIN {X 0,Y 319.892,Z 158.637,A -85,B 0,C 180,E1 -15383.693,E2 -15383.693} C_VEL
LIN {X 0,Y 319.71,Z 158.785,A -85,B 0,C 180,E1 -15385.548,E2 -15385.548} C_VEL
LIN {X 0,Y 321.096,Z 164.492,A -85,B 0,C 180,E1 -15387.373,E2 -15387.373} C_VEL
LIN {X 0,Y 328.177,Z 184.048,A -85,B 0,C 180,E1 -15388.371,E2 -15388.371} C_VEL
LIN {X 0,Y 330.204,Z 195.271,A -85,B 0,C 180,E1 -15388.78,E2 -15388.78} C_VEL
LIN {X 0,Y 328.293,Z 272.106,A -85,B 0,C 180,E1 -15390.498,E2 -15390.498} C_VEL
LIN {X 0,Y 327.636,Z 285.272,A -85,B 0,C 180,E1 -15391.037,E2 -15391.037} C_VEL
LIN {X 0,Y 326.876,Z 297.36,A -85,B 0,C 180,E1 -15391.771,E2 -15391.771} C_VEL
LIN {X 0,Y 325.861,Z 309.613,A -85,B 0,C 180,E1 -15392.781,E2 -15392.781} C_VEL
LIN {X 0,Y 324.606,Z 321.246,A -85,B 0,C 180,E1 -15394.027,E2 -15394.027} C_VEL
LIN {X 0,Y 323.328,Z 331.83,A -85,B 0,C 180,E1 -15395.457,E2 -15395.457} C_VEL
LIN {X 0,Y 322.224,Z 340.397,A -85,B 0,C 180,E1 -15396.89,E2 -15396.89} C_VEL
LIN {X 0,Y 320.877,Z 349.7,A -85,B 0,C 180,E1 -15398.819,E2 -15398.819} C_VEL
LIN {X 0,Y 319.886,Z 357.158,A -85,B 0,C 180,E1 -15400.763,E2 -15400.763} C_VEL
LIN {X 0,Y 319.071,Z 363.092,A -85,B 0,C 180,E1 -15402.724,E2 -15402.724} C_VEL
LIN {X 0,Y 318.511,Z 367.73,A -85,B 0,C 180,E1 -15404.699,E2 -15404.699} C_VEL
LIN {X 0,Y 318.073,Z 371.233,A -85,B 0,C 180,E1 -15406.693,E2 -15406.693} C_VEL
LIN {X 0,Y 317.835,Z 372.989,A -85,B 0,C 180,E1 -15408.048,E2 -15408.048} C_VEL
LIN {X 0,Y 317.695,Z 374.272,A -85,B 0,C 180,E1 -15409.38,E2 -15409.38} C_VEL
LIN {X 0,Y 317.62,Z 375.384,A -85,B 0,C 180,E1 -15411.672,E2 -15411.672} C_VEL
LIN {X 0,Y 317.668,Z 375.38,A -85,B 0,C 180,E1 -15413.467,E2 -15413.467} C_VEL
LIN {X 0,Y 317.794,Z 374.74,A -85,B 0,C 180,E1 -15414.948,E2 -15414.948} C_VEL
LIN {X 0,Y 317.939,Z 373.768,A -85,B 0,C 180,E1 -15416.238,E2 -15416.238} C_VEL
LIN {X 0,Y 318.31,Z 371.768,A -85,B 0,C 180,E1 -15417.976,E2 -15417.976} C_VEL
LIN {X 0,Y 318.912,Z 367.549,A -85,B 0,C 180,E1 -15420.455,E2 -15420.455} C_VEL
LIN {X 0,Y 319.748,Z 362.405,A -85,B 0,C 180,E1 -15422.582,E2 -15422.582} C_VEL
LIN {X 0,Y 320.863,Z 355.671,A -85,B 0,C 180,E1 -15424.715,E2 -15424.715} C_VEL
LIN {X 0,Y 322.091,Z 348.622,A -85,B 0,C 180,E1 -15426.483,E2 -15426.483} C_VEL
LIN {X 0,Y 323.448,Z 340.158,A -85,B 0,C 180,E1 -15428.204,E2 -15428.204} C_VEL
LIN {X 0,Y 324.983,Z 330.068,A -85,B 0,C 180,E1 -15429.841,E2 -15429.841} C_VEL
LIN {X 0,Y 326.465,Z 319.445,A -85,B 0,C 180,E1 -15431.22,E2 -15431.22} C_VEL
LIN {X 0,Y 327.707,Z 309.125,A -85,B 0,C 180,E1 -15432.289,E2 -15432.289} C_VEL
LIN {X 0,Y 328.76,Z 298.438,A -85,B 0,C 180,E1 -15433.163,E2 -15433.163} C_VEL
LIN {X 0,Y 329.729,Z 285.33,A -85,B 0,C 180,E1 -15433.957,E2 -15433.957} C_VEL
LIN {X 0,Y 330.373,Z 272.457,A -85,B 0,C 180,E1 -15434.482,E2 -15434.482} C_VEL
LIN {X 0,Y 331.196,Z 243.056,A -85,B 0,C 180,E1 -15435.16,E2 -15435.16} C_VEL
LIN {X 0,Y 330.756,Z 237.258,A -85,B 0,C 180,E1 -15435.338,E2 -15435.338} C_VEL
LIN {X 0,Y 326.158,Z 218.597,A -85,B 0,C 180,E1 -15436.19,E2 -15436.19} C_VEL
LIN {X 0,Y 325.642,Z 212.802,A -85,B 0,C 180,E1 -15436.38,E2 -15436.38} C_VEL
LIN {X 0,Y 326.066,Z 195.683,A -85,B 0,C 180,E1 -15436.773,E2 -15436.773} C_VEL
LIN {X 0,Y 324.915,Z 190.973,A -85,B 0,C 180,E1 -15436.998,E2 -15436.998} C_VEL
LIN {X 0,Y 318.245,Z 174.759,A -85,B 0,C 180,E1 -15438.053,E2 -15438.053} C_VEL
LIN {X 0,Y 313.972,Z 165.544,A -85,B 0,C 180,E1 -15438.73,E2 -15438.73} C_VEL
LIN {X 0,Y 312.532,Z 159.555,A -85,B 0,C 180,E1 -15440.847,E2 -15440.847} C_VEL
LIN {X 0,Y 312.529,Z 159.558,A -85,B 0,C 180,E1 -15444.221,E2 -15444.221} C_VEL
LIN {X 0,Y 312.501,Z 159.562,A -85,B 0,C 180,E1 -15447.335,E2 -15447.335} C_VEL
LIN {X 0,Y 312.55,Z 159.553,A -85,B 0,C 180,E1 -15451.277,E2 -15451.277} C_VEL
LIN {X 0,Y 312.584,Z 159.552,A -85,B 0,C 180,E1 -15454.712,E2 -15454.712} C_VEL
LIN {X 0,Y 312.586,Z 159.551,A -85,B 0,C 180,E1 -15457.53,E2 -15457.53} C_VEL
LIN {X 0,Y 312.588,Z 159.546,A -85,B 0,C 180,E1 -15461.655,E2 -15461.655} C_VEL
LIN {X 0,Y 312.685,Z 159.532,A -85,B 0,C 180,E1 -15465.687,E2 -15465.687} C_VEL
LIN {X 0,Y 312.686,Z 159.533,A -85,B 0,C 180,E1 -15469.642,E2 -15469.642} C_VEL
LIN {X 0,Y 312.8,Z 159.514,A -85,B 0,C 180,E1 -15472.254,E2 -15472.254} C_VEL
LIN {X 0,Y 312.702,Z 159.524,A -85,B 0,C 180,E1 -15474.843,E2 -15474.843} C_VEL
LIN {X 0,Y 312.932,Z 159.499,A -85,B 0,C 180,E1 -15477.427,E2 -15477.427} C_VEL
LIN {X 0,Y 313.052,Z 159.478,A -85,B 0,C 180,E1 -15480.001,E2 -15480.001} C_VEL
LIN {X 0,Y 312.907,Z 159.503,A -85,B 0,C 180,E1 -15482.576,E2 -15482.576} C_VEL
LIN {X 0,Y 312.844,Z 159.503,A -85,B 0,C 180,E1 -15486.45,E2 -15486.45} C_VEL
LIN {X 0,Y 312.752,Z 159.522,A -85,B 0,C 180,E1 -15489.051,E2 -15489.051} C_VEL
LIN {X 0,Y 312.634,Z 159.539,A -85,B 0,C 180,E1 -15492.992,E2 -15492.992} C_VEL
LIN {X 0,Y 312.613,Z 159.535,A -85,B 0,C 180,E1 -15495.652,E2 -15495.652} C_VEL
LIN {X 0,Y 312.537,Z 159.553,A -85,B 0,C 180,E1 -15499.714,E2 -15499.714} C_VEL
LIN {X 0,Y 312.516,Z 159.552,A -85,B 0,C 180,E1 -15502.776,E2 -15502.776} C_VEL
LIN {X 0,Y 312.485,Z 159.551,A -85,B 0,C 180,E1 -15506.733,E2 -15506.733} C_VEL
LIN {X 0,Y 312.497,Z 159.553,A -85,B 0,C 180,E1 -15509.656,E2 -15509.656} C_VEL
LIN {X 0,Y 312.522,Z 159.551,A -85,B 0,C 180,E1 -15513.689,E2 -15513.689} C_VEL
LIN {X 0,Y 312.511,Z 159.553,A -85,B 0,C 180,E1 -15517.388,E2 -15517.388} C_VEL
LIN {X 0,Y 312.442,Z 159.566,A -85,B 0,C 180,E1 -15520.718,E2 -15520.718} C_VEL
LIN {X 0,Y 312.452,Z 159.565,A -85,B 0,C 180,E1 -15524.211,E2 -15524.211} C_VEL
LIN {X 0,Y 312.456,Z 159.57,A -85,B 0,C 180,E1 -15527.926,E2 -15527.926} C_VEL
LIN {X 0,Y 312.479,Z 159.563,A -85,B 0,C 180,E1 -15531.925,E2 -15531.925} C_VEL
LIN {X 0,Y 312.534,Z 159.55,A -85,B 0,C 180,E1 -15534.221,E2 -15534.221} C_VEL
LIN {X 0,Y 312.543,Z 159.666,A -85,B 0,C 180,E1 -15535.952,E2 -15535.952} C_VEL
LIN {X 0,Y 315.195,Z 170.589,A -85,B 0,C 180,E1 -15539.469,E2 -15539.469} C_VEL
LIN {X 0,Y 317.329,Z 181.188,A -85,B 0,C 180,E1 -15542.659,E2 -15542.659} C_VEL
LIN {X 0,Y 317.825,Z 185.009,A -85,B 0,C 180,E1 -15543.699,E2 -15543.699} C_VEL
LIN {X 0,Y 321.483,Z 203.272,A -85,B 0,C 180,E1 -15544.522,E2 -15544.522} C_VEL
LIN {X 0,Y 324.661,Z 222.928,A -85,B 0,C 180,E1 -15545.311,E2 -15545.311} C_VEL
LIN {X 0,Y 325.332,Z 228.377,A -85,B 0,C 180,E1 -15545.507,E2 -15545.507} C_VEL
LIN {X 0,Y 323.603,Z 294.127,A -85,B 0,C 180,E1 -15547.03,E2 -15547.03} C_VEL
LIN {X 0,Y 322.623,Z 307.83,A -85,B 0,C 180,E1 -15547.591,E2 -15547.591} C_VEL
LIN {X 0,Y 321.389,Z 320.212,A -85,B 0,C 180,E1 -15548.345,E2 -15548.345} C_VEL
LIN {X 0,Y 320.123,Z 331.302,A -85,B 0,C 180,E1 -15549.267,E2 -15549.267} C_VEL
LIN {X 0,Y 318.441,Z 342.877,A -85,B 0,C 180,E1 -15550.5,E2 -15550.5} C_VEL
LIN {X 0,Y 316.762,Z 353.322,A -85,B 0,C 180,E1 -15551.904,E2 -15551.904} C_VEL
LIN {X 0,Y 315.329,Z 363.262,A -85,B 0,C 180,E1 -15553.596,E2 -15553.596} C_VEL
LIN {X 0,Y 313.953,Z 371.86,A -85,B 0,C 180,E1 -15555.414,E2 -15555.414} C_VEL
LIN {X 0,Y 312.597,Z 379.222,A -85,B 0,C 180,E1 -15557.338,E2 -15557.338} C_VEL
LIN {X 0,Y 311.639,Z 385.994,A -85,B 0,C 180,E1 -15559.606,E2 -15559.606} C_VEL
LIN {X 0,Y 311.121,Z 390.486,A -85,B 0,C 180,E1 -15561.557,E2 -15561.557} C_VEL
LIN {X 0,Y 310.822,Z 393.902,A -85,B 0,C 180,E1 -15563.509,E2 -15563.509} C_VEL
LIN {X 0,Y 310.717,Z 396.916,A -85,B 0,C 180,E1 -15566.109,E2 -15566.109} C_VEL
LIN {X 0,Y 310.701,Z 397.821,A -85,B 0,C 180,E1 -15567.407,E2 -15567.407} C_VEL
LIN {X 0,Y 310.701,Z 398.285,A -85,B 0,C 180,E1 -15568.704,E2 -15568.704} C_VEL
LIN {X 0,Y 310.761,Z 398.353,A -85,B 0,C 180,E1 -15570,E2 -15570} C_VEL
LIN {X 0,Y 310.712,Z 398.026,A -85,B 0,C 180,E1 -15571.296,E2 -15571.296} C_VEL
LIN {X 0,Y 310.703,Z 397.307,A -85,B 0,C 180,E1 -15572.593,E2 -15572.593} C_VEL
LIN {X 0,Y 310.718,Z 396.142,A -85,B 0,C 180,E1 -15573.891,E2 -15573.891} C_VEL
LIN {X 0,Y 310.727,Z 393.964,A -85,B 0,C 180,E1 -15575.614,E2 -15575.614} C_VEL
LIN {X 0,Y 310.984,Z 390.064,A -85,B 0,C 180,E1 -15577.793,E2 -15577.793} C_VEL
LIN {X 0,Y 311.389,Z 385.39,A -85,B 0,C 180,E1 -15579.746,E2 -15579.746} C_VEL
LIN {X 0,Y 312.191,Z 378.327,A -85,B 0,C 180,E1 -15582.019,E2 -15582.019} C_VEL
LIN {X 0,Y 313.299,Z 370.682,A -85,B 0,C 180,E1 -15583.955,E2 -15583.955} C_VEL
LIN {X 0,Y 314.541,Z 361.616,A -85,B 0,C 180,E1 -15585.782,E2 -15585.782} C_VEL
LIN {X 0,Y 315.801,Z 351.107,A -85,B 0,C 180,E1 -15587.484,E2 -15587.484} C_VEL
LIN {X 0,Y 317.297,Z 339.951,A -85,B 0,C 180,E1 -15588.902,E2 -15588.902} C_VEL
LIN {X 0,Y 318.592,Z 329.019,A -85,B 0,C 180,E1 -15589.994,E2 -15589.994} C_VEL
LIN {X 0,Y 319.816,Z 316.96,A -85,B 0,C 180,E1 -15590.922,E2 -15590.922} C_VEL
LIN {X 0,Y 320.846,Z 304.635,A -85,B 0,C 180,E1 -15591.609,E2 -15591.609} C_VEL
LIN {X 0,Y 321.478,Z 291.492,A -85,B 0,C 180,E1 -15592.085,E2 -15592.085} C_VEL
LIN {X 0,Y 322.832,Z 226.389,A -85,B 0,C 180,E1 -15593.575,E2 -15593.575} C_VEL
LIN {X 0,Y 317.146,Z 189.019,A -85,B 0,C 180,E1 -15594.901,E2 -15594.901} C_VEL
LIN {X 0,Y 316.612,Z 185.786,A -85,B 0,C 180,E1 -15595.033,E2 -15595.033} C_VEL
LIN {X 0,Y 316.992,Z 182.188,A -85,B 0,C 180,E1 -15595.969,E2 -15595.969} C_VEL
LIN {X 0,Y 315.683,Z 174.174,A -85,B 0,C 180,E1 -15598.235,E2 -15598.235} C_VEL
LIN {X 0,Y 313.32,Z 163.065,A -85,B 0,C 180,E1 -15601.528,E2 -15601.528} C_VEL
LIN {X 0,Y 312.554,Z 159.554,A -85,B 0,C 180,E1 -15602.661,E2 -15602.661} C_VEL
LIN {X 0,Y 312.539,Z 159.554,A -85,B 0,C 180,E1 -15605.949,E2 -15605.949} C_VEL
LIN {X 0,Y 312.459,Z 159.563,A -85,B 0,C 180,E1 -15610.114,E2 -15610.114} C_VEL
LIN {X 0,Y 312.461,Z 159.562,A -85,B 0,C 180,E1 -15613.964,E2 -15613.964} C_VEL
LIN {X 0,Y 312.46,Z 159.562,A -85,B 0,C 180,E1 -15617.924,E2 -15617.924} C_VEL
LIN {X 0,Y 312.488,Z 159.558,A -85,B 0,C 180,E1 -15621.922,E2 -15621.922} C_VEL
LIN {X 0,Y 312.535,Z 159.552,A -85,B 0,C 180,E1 -15624.22,E2 -15624.22} C_VEL
LIN {X 0,Y 312.506,Z 159.558,A -85,B 0,C 180,E1 -15627.333,E2 -15627.333} C_VEL
LIN {X 0,Y 312.511,Z 159.557,A -85,B 0,C 180,E1 -15631.291,E2 -15631.291} C_VEL
LIN {X 0,Y 312.552,Z 159.554,A -85,B 0,C 180,E1 -15634.707,E2 -15634.707} C_VEL
LIN {X 0,Y 312.522,Z 159.557,A -85,B 0,C 180,E1 -15638.911,E2 -15638.911} C_VEL
LIN {X 0,Y 312.556,Z 159.549,A -85,B 0,C 180,E1 -15641.65,E2 -15641.65} C_VEL
LIN {X 0,Y 312.656,Z 159.536,A -85,B 0,C 180,E1 -15645.683,E2 -15645.683} C_VEL
LIN {X 0,Y 312.69,Z 159.531,A -85,B 0,C 180,E1 -15649.64,E2 -15649.64} C_VEL
LIN {X 0,Y 312.8,Z 159.517,A -85,B 0,C 180,E1 -15652.251,E2 -15652.251} C_VEL
LIN {X 0,Y 312.692,Z 159.532,A -85,B 0,C 180,E1 -15654.841,E2 -15654.841} C_VEL
LIN {X 0,Y 312.971,Z 159.498,A -85,B 0,C 180,E1 -15658.712,E2 -15658.712} C_VEL
LIN {X 0,Y 312.971,Z 159.494,A -85,B 0,C 180,E1 -15661.286,E2 -15661.286} C_VEL
LIN {X 0,Y 312.689,Z 159.528,A -85,B 0,C 180,E1 -15665.157,E2 -15665.157} C_VEL
LIN {X 0,Y 312.798,Z 159.52,A -85,B 0,C 180,E1 -15667.746,E2 -15667.746} C_VEL
LIN {X 0,Y 312.662,Z 159.538,A -85,B 0,C 180,E1 -15671.67,E2 -15671.67} C_VEL
LIN {X 0,Y 312.615,Z 159.536,A -85,B 0,C 180,E1 -15674.826,E2 -15674.826} C_VEL
LIN {X 0,Y 312.536,Z 159.551,A -85,B 0,C 180,E1 -15679.184,E2 -15679.184} C_VEL
LIN {X 0,Y 312.514,Z 159.554,A -85,B 0,C 180,E1 -15682.773,E2 -15682.773} C_VEL
LIN {X 0,Y 312.482,Z 159.553,A -85,B 0,C 180,E1 -15686.731,E2 -15686.731} C_VEL
LIN {X 0,Y 312.468,Z 159.563,A -85,B 0,C 180,E1 -15689.657,E2 -15689.657} C_VEL
LIN {X 0,Y 312.518,Z 159.556,A -85,B 0,C 180,E1 -15693.687,E2 -15693.687} C_VEL
LIN {X 0,Y 312.508,Z 159.554,A -85,B 0,C 180,E1 -15697.386,E2 -15697.386} C_VEL
LIN {X 0,Y 312.438,Z 159.563,A -85,B 0,C 180,E1 -15700.716,E2 -15700.716} C_VEL
LIN {X 0,Y 312.447,Z 159.563,A -85,B 0,C 180,E1 -15704.209,E2 -15704.209} C_VEL
LIN {X 0,Y 312.451,Z 159.56,A -85,B 0,C 180,E1 -15707.924,E2 -15707.924} C_VEL
LIN {X 0,Y 312.479,Z 159.559,A -85,B 0,C 180,E1 -15711.921,E2 -15711.921} C_VEL
LIN {X 0,Y 312.525,Z 159.552,A -85,B 0,C 180,E1 -15714.219,E2 -15714.219} C_VEL
LIN {X 0,Y 312.496,Z 159.558,A -85,B 0,C 180,E1 -15717.332,E2 -15717.332} C_VEL
LIN {X 0,Y 312.499,Z 159.556,A -85,B 0,C 180,E1 -15721.291,E2 -15721.291} C_VEL
LIN {X 0,Y 312.51,Z 159.559,A -85,B 0,C 180,E1 -15724.704,E2 -15724.704} C_VEL
LIN {X 0,Y 312.532,Z 159.55,A -85,B 0,C 180,E1 -15727.524,E2 -15727.524} C_VEL
LIN {X 0,Y 312.544,Z 159.551,A -85,B 0,C 180,E1 -15731.65,E2 -15731.65} C_VEL
LIN {X 0,Y 312.644,Z 159.538,A -85,B 0,C 180,E1 -15735.684,E2 -15735.684} C_VEL
LIN {X 0,Y 312.677,Z 159.534,A -85,B 0,C 180,E1 -15739.641,E2 -15739.641} C_VEL
LIN {X 0,Y 312.789,Z 159.525,A -85,B 0,C 180,E1 -15742.252,E2 -15742.252} C_VEL
LIN {X 0,Y 312.693,Z 159.547,A -85,B 0,C 180,E1 -15745.124,E2 -15745.124} C_VEL
LIN {X 0,Y 313.905,Z 164.942,A -85,B 0,C 180,E1 -15746.838,E2 -15746.838} C_VEL
LIN {X 0,Y 320.757,Z 183.271,A -85,B 0,C 180,E1 -15747.817,E2 -15747.817} C_VEL
LIN {X 0,Y 322.419,Z 188.995,A -85,B 0,C 180,E1 -15748.078,E2 -15748.078} C_VEL
LIN {X 0,Y 323.615,Z 195.635,A -85,B 0,C 180,E1 -15748.325,E2 -15748.325} C_VEL
LIN {X 0,Y 321.634,Z 272.464,A -85,B 0,C 180,E1 -15750.078,E2 -15750.078} C_VEL
LIN {X 0,Y 320.949,Z 285.6,A -85,B 0,C 180,E1 -15750.627,E2 -15750.627} C_VEL
LIN {X 0,Y 320.116,Z 298.241,A -85,B 0,C 180,E1 -15751.415,E2 -15751.415} C_VEL
LIN {X 0,Y 319.145,Z 309.511,A -85,B 0,C 180,E1 -15752.366,E2 -15752.366} C_VEL
LIN {X 0,Y 317.811,Z 321.286,A -85,B 0,C 180,E1 -15753.645,E2 -15753.645} C_VEL
LIN {X 0,Y 316.488,Z 331.86,A -85,B 0,C 180,E1 -15755.096,E2 -15755.096} C_VEL
LIN {X 0,Y 315.217,Z 341.312,A -85,B 0,C 180,E1 -15756.722,E2 -15756.722} C_VEL
LIN {X 0,Y 313.861,Z 350.501,A -85,B 0,C 180,E1 -15758.693,E2 -15758.693} C_VEL
LIN {X 0,Y 312.823,Z 357.848,A -85,B 0,C 180,E1 -15760.681,E2 -15760.681} C_VEL
LIN {X 0,Y 312.108,Z 362.816,A -85,B 0,C 180,E1 -15762.352,E2 -15762.352} C_VEL
LIN {X 0,Y 311.501,Z 367.59,A -85,B 0,C 180,E1 -15764.37,E2 -15764.37} C_VEL
LIN {X 0,Y 311.032,Z 371.206,A -85,B 0,C 180,E1 -15766.406,E2 -15766.406} C_VEL
LIN {X 0,Y 310.695,Z 373.746,A -85,B 0,C 180,E1 -15768.462,E2 -15768.462} C_VEL
LIN {X 0,Y 310.58,Z 374.845,A -85,B 0,C 180,E1 -15769.842,E2 -15769.842} C_VEL
LIN {X 0,Y 310.532,Z 375.67,A -85,B 0,C 180,E1 -15771.891,E2 -15771.891} C_VEL
LIN {X 0,Y 310.621,Z 375.475,A -85,B 0,C 180,E1 -15774.033,E2 -15774.033} C_VEL
LIN {X 0,Y 310.764,Z 374.766,A -85,B 0,C 180,E1 -15775.448,E2 -15775.448} C_VEL
LIN {X 0,Y 310.957,Z 373.554,A -85,B 0,C 180,E1 -15776.873,E2 -15776.873} C_VEL
LIN {X 0,Y 311.443,Z 370.771,A -85,B 0,C 180,E1 -15779.023,E2 -15779.023} C_VEL
LIN {X 0,Y 312.105,Z 366.723,A -85,B 0,C 180,E1 -15781.192,E2 -15781.192} C_VEL
LIN {X 0,Y 313.024,Z 361.522,A -85,B 0,C 180,E1 -15783.276,E2 -15783.276} C_VEL
LIN {X 0,Y 314.066,Z 355.451,A -85,B 0,C 180,E1 -15785.185,E2 -15785.185} C_VEL
LIN {X 0,Y 315.371,Z 348.288,A -85,B 0,C 180,E1 -15786.991,E2 -15786.991} C_VEL
LIN {X 0,Y 316.961,Z 338.698,A -85,B 0,C 180,E1 -15788.916,E2 -15788.916} C_VEL
LIN {X 0,Y 318.481,Z 329.417,A -85,B 0,C 180,E1 -15790.408,E2 -15790.408} C_VEL
LIN {X 0,Y 320.012,Z 318.461,A -85,B 0,C 180,E1 -15791.825,E2 -15791.825} C_VEL
LIN {X 0,Y 321.339,Z 307.884,A -85,B 0,C 180,E1 -15792.901,E2 -15792.901} C_VEL
LIN {X 0,Y 322.6,Z 294.914,A -85,B 0,C 180,E1 -15793.919,E2 -15793.919} C_VEL
LIN {X 0,Y 323.439,Z 282.448,A -85,B 0,C 180,E1 -15794.624,E2 -15794.624} C_VEL
LIN {X 0,Y 324.119,Z 268.744,A -85,B 0,C 180,E1 -15795.108,E2 -15795.108} C_VEL
LIN {X 0,Y 325.642,Z 212.802,A -85,B 0,C 180,E1 -15796.38,E2 -15796.38} C_VEL
LIN {X 0,Y 325.004,Z 207.655,A -85,B 0,C 180,E1 -15796.567,E2 -15796.567} C_VEL
LIN {X 0,Y 323.389,Z 202.809,A -85,B 0,C 180,E1 -15796.838,E2 -15796.838} C_VEL
LIN {X 0,Y 318.932,Z 193.583,A -85,B 0,C 180,E1 -15797.495,E2 -15797.495} C_VEL
LIN {X 0,Y 312.497,Z 178.001,A -85,B 0,C 180,E1 -15798.546,E2 -15798.546} C_VEL
LIN {X 0,Y 306.838,Z 165.772,A -85,B 0,C 180,E1 -15799.511,E2 -15799.511} C_VEL
LIN {X 0,Y 305.492,Z 160.434,A -85,B 0,C 180,E1 -15801.461,E2 -15801.461} C_VEL
